# B&R Automation Studio project NewPendant_NG4_11_05_25A (part 19)

```c
					TVL_ROT_Param_Set[i].pEncoder = &AxisCh[TML_AX_TVL].curPos;
					TVL_ROT_Param_Set[i].pHomePos = &OLD_MTR_POS[TVL_ENC_HOME];
					TVL_ROT_Param_Set[i].EncPerTick = m->pCfg->HeadCfg.TVL.EncPerTick;
					TVL_ROT_Param_Set[i].EncDir = m->pCfg->HeadCfg.TVL.Enc_Dir;
					TVL_ROT_Param_Set[i].TicksAtHighVel = 3;

				break;

			}
		}

		for(i=0 ; i < 1 ; i++){

			switch(i){

				case 0:

					strcpy(Process[m->pCfg->HeadCfg.INDX.PROC_Indx].Name , "INDX");
					INDEX_Param_Set[i].pPrc = &Process[m->pCfg->HeadCfg.INDX.PROC_Indx];
					Process[m->pCfg->HeadCfg.INDX.PROC_Indx].Disable = 1;

				break;

			}

		}

	return 1;

}

DINT Configure_OMEGA_16INCH_HP_ENCODER(MASTER_typ *m  , UINT headType ){

}

/////////////////////////////////////////////////////////////

void ParametrAssignToPointers(MASTER_typ *m  , UINT indx){
int i;
CurCfg_typ *c;
Cfg_typ *cfg;
CurCalib_typ *calib;
DINT headType;

	if(!m)
		return;

	if(!m->pCurCfg)
		return;

	if(!m->pCalib)
		return;

	if(!m->pCalib->GenSetup)
		return;

	if(!m->pCfg)
		return;

	cfg = m->pCfg;

	c = m->pCurCfg;

	 headType = m->pCalib->GenSetup[SETUP_HEAD_SETUP];

	for(i=0 ; i < 1; i++){

		switch(i){

			case 0:

				//strcpy(Process[PROC_TIG_PS].Name , "TIG PS");

				if(c->Param[parTIG_StartDly].segmYes)
						PS_Param_Set[i].pStartDly		= &c->Param[parTIG_StartDly].val[indx];
				else 	PS_Param_Set[i].pStartDly		= &c->Param[parTIG_StartDly].val[0];

				if(c->Param[parTIG_StopDly].segmYes)
						PS_Param_Set[i].pStopDly		= &c->Param[parTIG_StopDly].val[indx];
				else		PS_Param_Set[i].pStopDly		= &c->Param[parTIG_StopDly].val[0];

				if(c->Param[parTIG_RampUp].segmYes)
						PS_Param_Set[i].pRampUp			= &c->Param[parTIG_RampUp].val[indx];
				else		PS_Param_Set[i].pRampUp			= &c->Param[parTIG_RampUp].val[0];

				if(c->Param[parTIG_RampDwn].segmYes)
						PS_Param_Set[i].pRampDwn		= &c->Param[parTIG_RampDwn].val[indx];
				else	PS_Param_Set[i].pRampDwn		= &c->Param[parTIG_RampDwn].val[0];

				if(c->Param[parTIG_AmpSP].segmYes)
						PS_Param_Set[i].pAmpSP			= &c->Param[parTIG_AmpSP].val[indx];
				else	PS_Param_Set[i].pAmpSP			= &c->Param[parTIG_AmpSP].val[0];

				if(c->Param[parTIG_AmpInSP].segmYes)
						PS_Param_Set[i].pAmpInSP		= &c->Param[parTIG_AmpInSP].val[indx];
				else	PS_Param_Set[i].pAmpInSP		= &c->Param[parTIG_AmpInSP].val[0];

				if(c->Param[parTIG_AmpOutSP].segmYes)
						PS_Param_Set[i].pAmpOutSP		= &c->Param[parTIG_AmpOutSP].val[indx];
				else	PS_Param_Set[i].pAmpOutSP		= &c->Param[parTIG_AmpOutSP].val[0];

				if(c->Param[parTIG_BackAmp].segmYes)
						PS_Param_Set[i].pBackAmp		= &c->Param[parTIG_BackAmp].val[indx];
				else		PS_Param_Set[i].pBackAmp 		= &c->Param[parTIG_BackAmp].val[0];

				if(c->Param[parTIG_StartAmp].segmYes)
						PS_Param_Set[i].pStartAmp		= &c->Param[parTIG_StartAmp].val[indx];
				else		PS_Param_Set[i].pStartAmp		= &c->Param[parTIG_StartAmp].val[0];

				if(c->Param[parTIG_EndAmp].segmYes)
						PS_Param_Set[i].pEndAmp			= &c->Param[parTIG_EndAmp].val[indx];
				else		PS_Param_Set[i].pEndAmp			= &c->Param[parTIG_EndAmp].val[0];

				if(c->Param[parTIG_AmpSP_Boost].segmYes)
						PS_Param_Set[i].pAmpBoost 		= &c->Param[parTIG_AmpSP_Boost].val[indx];
				else	PS_Param_Set[i].pAmpBoost 			= &c->Param[parTIG_AmpSP_Boost].val[0];

				if(c->Param_ENUM[parENUM_TIG_Mode].segmYes)
						PS_Param_Set[i].pMode			= &c->Param_ENUM[parENUM_TIG_Mode].val[indx];
				else 	PS_Param_Set[i].pMode			= &c->Param_ENUM[parENUM_TIG_Mode].val[0];

				if(c->Param[parTIG_PulseFreq].segmYes)
						PS_Param_Set[i].pPulseFreq 		= &c->Param[parTIG_PulseFreq].val[indx];
				else		PS_Param_Set[i].pPulseFreq 		= &c->Param[parTIG_PulseFreq].val[0];

				if(c->Param[parTIG_PulseWidth].segmYes)
						PS_Param_Set[i].pPulseWidth 		= &c->Param[parTIG_PulseWidth].val[indx];
				else		PS_Param_Set[i].pPulseWidth 		= &c->Param[parTIG_PulseWidth].val[0];

				if(c->Param[parTIG_Boost1].segmYes)
						PS_Param_Set[i].pBoost1 		= &c->Param[parTIG_Boost1].val[indx];
				else	PS_Param_Set[i].pBoost1 		= &c->Param[parTIG_Boost1].val[0];

				if(c->Param[parTIG_Boost2].segmYes)
						PS_Param_Set[i].pBoost2 		= &c->Param[parTIG_Boost2].val[indx];
				else	PS_Param_Set[i].pBoost2 		= &c->Param[parTIG_Boost2].val[0];

				if(c->Param[parCONTIN_TIG_RampDwn].segmYes)
						PS_Param_Set[i].pContin_RampDwn 		= &c->Param[parCONTIN_TIG_RampDwn].val[indx];
				else	PS_Param_Set[i].pContin_RampDwn 		= &c->Param[parCONTIN_TIG_RampDwn].val[0];

				if(c->Param[parCONTIN_TIG_RampUp].segmYes)
						PS_Param_Set[i].pContin_RampUp 		= &c->Param[parCONTIN_TIG_RampUp].val[indx];
				else	PS_Param_Set[i].pContin_RampUp 		= &c->Param[parCONTIN_TIG_RampUp].val[0];

				if(c->Param[parCONTIN_TIG_Dwell].segmYes)
						PS_Param_Set[i].pContin_Dwell 		= &c->Param[parCONTIN_TIG_Dwell].val[indx];
				else	PS_Param_Set[i].pContin_Dwell 		= &c->Param[parCONTIN_TIG_Dwell].val[0];

				if(c->Param[parCONTIN_TIG_Percent].segmYes)
						PS_Param_Set[i].pContin_Amp_Reduce 		= &c->Param[parCONTIN_TIG_Percent].val[indx];
				else	PS_Param_Set[i].pContin_Amp_Reduce 		= &c->Param[parCONTIN_TIG_Percent].val[0];

			break;

		}

	}

	for(i=0 ; i < 1 ; i++){

		switch(i){

			case 0:

				strcpy(Process[PROC_AVC].Name , "AVC");

				if(c->Param[parAVC_TouchVolt].segmYes)
						AVC_Param_Set[i].pTouchVolt 		= &c->Param[parAVC_TouchVolt].val[indx];
				else 	AVC_Param_Set[i].pTouchVolt 		= &c->Param[parAVC_TouchVolt].val[0];

				if(c->Param[parAVC_TouchTm].segmYes)
						AVC_Param_Set[i].pTouchTm 			= &c->Param[parAVC_TouchTm].val[indx];
				else 	AVC_Param_Set[i].pTouchTm 			= &c->Param[parAVC_TouchTm].val[0];

				if(c->Param[parAVC_TRetractTm].segmYes)
						AVC_Param_Set[i].pRetractTm 		= &c->Param[parAVC_TRetractTm].val[indx];
				else 	AVC_Param_Set[i].pRetractTm 		= &c->Param[parAVC_TRetractTm].val[0];

				if(c->Param[parAVC_TouchRepeat].segmYes)
						AVC_Param_Set[i].pTouchRepeat 		= &c->Param[parAVC_TouchRepeat].val[indx];
				else 	AVC_Param_Set[i].pTouchRepeat 		= &c->Param[parAVC_TouchRepeat].val[0];

				if(c->Param[parAVC_VoltSP].segmYes)
						AVC_Param_Set[i].pVoltSP 			= &c->Param[parAVC_VoltSP].val[indx];
				else 	AVC_Param_Set[i].pVoltSP 			= &c->Param[parAVC_VoltSP].val[0];

				if(c->Param[parAVC_VoltInSP].segmYes)
						AVC_Param_Set[i].pVoltInSP 			= &c->Param[parAVC_VoltInSP].val[indx];
				else 	AVC_Param_Set[i].pVoltInSP 			= &c->Param[parAVC_VoltInSP].val[0];

				if(c->Param[parAVC_VoltOutSP].segmYes)
						AVC_Param_Set[i].pVoltOutSP 		= &c->Param[parAVC_VoltOutSP].val[indx];
				else 	AVC_Param_Set[i].pVoltOutSP 		= &c->Param[parAVC_VoltOutSP].val[0];

				if(c->Param[parAVC_VoltBackSP].segmYes)
						AVC_Param_Set[i].pBkgVoltSP			= &c->Param[parAVC_VoltBackSP].val[indx];
				else 	AVC_Param_Set[i].pBkgVoltSP 		= &c->Param[parAVC_VoltBackSP].val[0];

				if(c->Param[parAVC_VSPTmOut].segmYes)
						AVC_Param_Set[i].pVoltSPTimeOut 	= &c->Param[parAVC_VSPTmOut].val[indx];
				else 	AVC_Param_Set[i].pVoltSPTimeOut 	= &c->Param[parAVC_VSPTmOut].val[0];

				if(c->Param[parAVC_TouchVel].segmYes)
						AVC_Param_Set[i].pTouchVel 			= &c->Param[parAVC_TouchVel].val[indx];
				else 	AVC_Param_Set[i].pTouchVel 			= &c->Param[parAVC_TouchVel].val[0];

				if(c->Param[parAVC_ToSPVel].segmYes)
						AVC_Param_Set[i].pToSPVel 			= &c->Param[parAVC_ToSPVel].val[indx];
				else 	AVC_Param_Set[i].pToSPVel 			= &c->Param[parAVC_ToSPVel].val[0];

				if(c->Param[parAVC_LU_TM].segmYes)
						AVC_Param_Set[i].pLU_Tm 			= &c->Param[parAVC_LU_TM].val[indx];
				else 	AVC_Param_Set[i].pLU_Tm 			= &c->Param[parAVC_LU_TM].val[0];

				if(c->Param[parAVC_KissTm].segmYes)
						AVC_Param_Set[i].pKiss_Tm 			= &c->Param[parAVC_KissTm].val[indx];
				else 	AVC_Param_Set[i].pKiss_Tm 			= &c->Param[parAVC_KissTm].val[0];

				if(c->Param[parAVC_VoltFinal].segmYes)
						AVC_Param_Set[i].pFinalVolt 		= &c->Param[parAVC_VoltFinal].val[indx];
				else 	AVC_Param_Set[i].pFinalVolt 		= &c->Param[parAVC_VoltFinal].val[0];

				if(c->Param[parAVC_DownSlope].segmYes)
						AVC_Param_Set[i].pRampDwn 		= &c->Param[parAVC_DownSlope].val[indx];
				else 	AVC_Param_Set[i].pRampDwn 		= &c->Param[parAVC_DownSlope].val[0];

				if(c->Param[parAVC_HoldTm].segmYes)
						AVC_Param_Set[i].pHoldTm 			= &c->Param[parAVC_HoldTm].val[indx];
				else 	AVC_Param_Set[i].pHoldTm 			= &c->Param[parAVC_HoldTm].val[0];

				if(c->Param[parAVC_GoBackTm].segmYes)
						AVC_Param_Set[i].pGoBackTm 			= &c->Param[parAVC_GoBackTm].val[indx];
				else 	AVC_Param_Set[i].pGoBackTm 			= &c->Param[parAVC_GoBackTm].val[0];

				if(c->Param[parAVC_StartDly].segmYes)
						AVC_Param_Set[i].pStartDly 			= &c->Param[parAVC_StartDly].val[indx];
				else 	AVC_Param_Set[i].pStartDly 			= &c->Param[parAVC_StartDly].val[0];

				if(c->Param[parAVC_StopDly].segmYes)
						AVC_Param_Set[i].pStopDly			= &c->Param[parAVC_StopDly].val[indx];
				else 	AVC_Param_Set[i].pStopDly 			= &c->Param[parAVC_StopDly].val[0];

				if(c->Param[parAVC_VoltInit].segmYes)
						AVC_Param_Set[i].pVoltInit			= &c->Param[parAVC_VoltInit].val[indx];
				else 	AVC_Param_Set[i].pVoltInit 			= &c->Param[parAVC_VoltInit].val[0];

				if(c->Param[parAVC_Upslope].segmYes)
						AVC_Param_Set[i].pRampUp 			= &c->Param[parAVC_Upslope].val[indx];
				else 	AVC_Param_Set[i].pRampUp 			= &c->Param[parAVC_Upslope].val[0];

				if(c->Param[parAVC_MaxVoltError].segmYes)
						AVC_Param_Set[i].pMaxVolrError 		= &c->Param[parAVC_MaxVoltError].val[indx];
				else 	AVC_Param_Set[i].pMaxVolrError 		= &c->Param[parAVC_MaxVoltError].val[0];

				if(c->Param[parAVC_Limits_Mask_Tm].segmYes)
						AVC_Param_Set[i].pLimitsFilterTm 	= &c->Param[parAVC_Limits_Mask_Tm].val[indx];
				else 	AVC_Param_Set[i].pLimitsFilterTm 	= &c->Param[parAVC_Limits_Mask_Tm].val[0];

				if(c->Param[parAVC_JogSpeedDirCntrl].segmYes)
						AVC_Param_Set[i].pJogSpeedDirCntrl	= &c->Param[parAVC_JogSpeedDirCntrl].val[indx];
				else 	AVC_Param_Set[i].pJogSpeedDirCntrl	= &c->Param[parAVC_JogSpeedDirCntrl].val[0];

				if(c->Param[parAVC_LiftSpeedDirCntrl].segmYes)
						AVC_Param_Set[i].pLiftSpeedDirCntrl	= &c->Param[parAVC_LiftSpeedDirCntrl].val[indx];
				else 	AVC_Param_Set[i].pLiftSpeedDirCntrl	= &c->Param[parAVC_LiftSpeedDirCntrl].val[0];

				if(c->Param_ENUM[parENUM_AVC_Mode].segmYes)
						AVC_Param_Set[i].pMode				= &c->Param_ENUM[parENUM_AVC_Mode].val[indx];
				else 	AVC_Param_Set[i].pMode				= &c->Param_ENUM[parENUM_AVC_Mode].val[0];

				if(c->Param[parAVC_LiftSpeedDirCntrl].segmYes)
						AVC_Param_Set[i].pJogSpeedDirCntrl	= &c->Param[parAVC_JogSpeedDirCntrl].val[indx];
				else 	AVC_Param_Set[i].pJogSpeedDirCntrl	= &c->Param[parAVC_JogSpeedDirCntrl].val[0];

				if(c->Param[parAVC_DB_Window].segmYes)
						AVC_Param_Set[i].pBB_Window 	= &c->Param[parAVC_DB_Window].val[indx];
				else 	AVC_Param_Set[i].pBB_Window		= &c->Param[parAVC_DB_Window].val[0];

				if(c->Param[parAVC_BB_Vel].segmYes)
						AVC_Param_Set[i].pBB_Vel		= &c->Param[parAVC_BB_Vel].val[indx];
				else 	AVC_Param_Set[i].pBB_Vel 	= &c->Param[parAVC_BB_Vel].val[0];

				if(c->Param[parAVC_BB_Gain].segmYes)
						AVC_Param_Set[i].pBB_Gain	= &c->Param[parAVC_BB_Gain].val[indx];
				else 	AVC_Param_Set[i].pBB_Gain 	= &c->Param[parAVC_BB_Gain].val[0];

				if(c->Param[parAVC_BB_Integr].segmYes)
						AVC_Param_Set[i].pBB_Integr	= &c->Param[parAVC_BB_Integr].val[indx];
				else 	AVC_Param_Set[i].pBB_Integr 	= &c->Param[parAVC_BB_Integr].val[0];

				if(c->Param[parAVC_Boost1].segmYes)
						AVC_Param_Set[i].pBoost1	= &c->Param[parAVC_Boost1].val[indx];
				else 	AVC_Param_Set[i].pBoost1 	= &c->Param[parAVC_Boost1].val[0];

				if(c->Param[parAVC_Boost2].segmYes)
						AVC_Param_Set[i].pBoost2	= &c->Param[parAVC_Boost2].val[indx];
				else 	AVC_Param_Set[i].pBoost2 	= &c->Param[parAVC_Boost2].val[0];

			break;

		}
	}

	for(i=0 ; i < 1 ; i++){

		switch(i){

			case 0:

				if(c->Param[parWRST_JogSpeedDirCntrl].segmYes)
						WRST_TML_Param_Set[i].pJogSpeedDirCntrl		= &c->Param[parWRST_JogSpeedDirCntrl].val[indx];
				else 	WRST_TML_Param_Set[i].pJogSpeedDirCntrl		= &c->Param[parWRST_JogSpeedDirCntrl].val[0];

				if(c->Param[parTVL_POS_OFFSET].segmYes)
						WRST_TML_Param_Set[i].pTVL_Pos_Offset 	= &c->Param[parTVL_POS_OFFSET].val[indx];
				else	WRST_TML_Param_Set[i].pTVL_Pos_Offset 	= &c->Param[parTVL_POS_OFFSET].val[0];

				if(c->Param[parTVL_POS_PREDICT].segmYes)
						WRST_TML_Param_Set[i].pTVL_Pos_Predict 	= &c->Param[parTVL_POS_PREDICT].val[indx];
				else	WRST_TML_Param_Set[i].pTVL_Pos_Predict 	= &c->Param[parTVL_POS_PREDICT].val[0];

				if(c->Param[parGEN_Radius].segmYes)
						WRST_TML_Param_Set[i].pRadius		= &c->Param[parGEN_Radius].val[indx];
				else 	WRST_TML_Param_Set[i].pRadius		= &c->Param[parGEN_Radius].val[0];

				if(c->Param[parGEN_RadSpeed_Boost].segmYes)
						WRST_TML_Param_Set[i].pRadSpeed_Boost		= &c->Param[parGEN_RadSpeed_Boost].val[indx];
				else 	WRST_TML_Param_Set[i].pRadSpeed_Boost		= &c->Param[parGEN_RadSpeed_Boost].val[0];

			break;

		}
	}

	for(i=0 ; i < 1 ; i++){

		switch(i){

			case 0:

				strcpy(Process[PROC_OSC].Name , "OSC");

				if(c->Param[parOSC_StartDly].segmYes)
						OSC_TML_Param_Set[i].pStartDly		= &c->Param[parOSC_StartDly].val[indx];
				else 	OSC_TML_Param_Set[i].pStartDly		= &c->Param[parOSC_StartDly].val[0];

				if(c->Param[parOSC_RampUp].segmYes)
						OSC_TML_Param_Set[i].pRampUp		= &c->Param[parOSC_RampUp].val[indx];
				else 	OSC_TML_Param_Set[i].pRampUp		= &c->Param[parOSC_RampUp].val[0];

				if(c->Param[parOSC_Amplit].segmYes)
						OSC_TML_Param_Set[i].pPrimAmpl		= &c->Param[parOSC_Amplit].val[indx];
				else 	OSC_TML_Param_Set[i].pPrimAmpl		= &c->Param[parOSC_Amplit].val[0];

				if(c->Param[parOSC_InitAmplit].segmYes)
						OSC_TML_Param_Set[i].pInitAmpl		= &c->Param[parOSC_InitAmplit].val[indx];
				else	OSC_TML_Param_Set[i].pInitAmpl		= &c->Param[parOSC_InitAmplit].val[0];

				if(c->Param[parOSC_FinalAmplit].segmYes)
						OSC_TML_Param_Set[i].pFinalAmpl		= &c->Param[parOSC_FinalAmplit].val[indx];
				else	OSC_TML_Param_Set[i].pFinalAmpl		= &c->Param[parOSC_FinalAmplit].val[0];

				if(c->Param[parOSC_StopDly].segmYes)
						OSC_TML_Param_Set[i].pStopDly		= &c->Param[parOSC_StopDly].val[indx];
				else 	OSC_TML_Param_Set[i].pStopDly		= &c->Param[parOSC_StopDly].val[0];

				if(c->Param[parOSC_RampDwn].segmYes)
						OSC_TML_Param_Set[i].pRampDwn		= &c->Param[parOSC_RampDwn].val[indx];
				else 	OSC_TML_Param_Set[i].pRampDwn		= &c->Param[parOSC_RampDwn].val[0];

				if(c->Param[parOSC_RampUpdate].segmYes)
						OSC_TML_Param_Set[i].pRampUpdate	= &c->Param[parOSC_RampUpdate].val[indx];
				else 	OSC_TML_Param_Set[i].pRampUpdate	= &c->Param[parOSC_RampUpdate].val[0];

				if(c->Param[parOSC_Excur].segmYes)
						OSC_TML_Param_Set[i].pFreq			= &c->Param[parOSC_Excur].val[indx];
				else 	OSC_TML_Param_Set[i].pFreq			= &c->Param[parOSC_Excur].val[0];

				if(cfg->HeadCfg.OSC.DwellDir > 0){

					if(c->Param[parOSC_Dwell_In].segmYes)
						OSC_TML_Param_Set[i].pDwell_In		= &c->Param[parOSC_Dwell_Out].val[indx];
					else	OSC_TML_Param_Set[i].pDwell_In		= &c->Param[parOSC_Dwell_Out].val[0];

					if(c->Param[parOSC_Dwell_Out].segmYes)
						OSC_TML_Param_Set[i].pDwell_Out 	= &c->Param[parOSC_Dwell_In].val[indx];
					else	OSC_TML_Param_Set[i].pDwell_Out 	= &c->Param[parOSC_Dwell_In].val[0];

				}
				else {

					if(c->Param[parOSC_Dwell_In].segmYes)
							OSC_TML_Param_Set[i].pDwell_In		= &c->Param[parOSC_Dwell_In].val[indx];
					else	OSC_TML_Param_Set[i].pDwell_In		= &c->Param[parOSC_Dwell_In].val[0];

					if(c->Param[parOSC_Dwell_Out].segmYes)
							OSC_TML_Param_Set[i].pDwell_Out 	= &c->Param[parOSC_Dwell_Out].val[indx];
					else	OSC_TML_Param_Set[i].pDwell_Out 	= &c->Param[parOSC_Dwell_Out].val[0];

				}

				if(c->Param_ENUM[parENUM_OSC_CAM].segmYes)
						OSC_TML_Param_Set[i].pCamType		= &c->Param_ENUM[parENUM_OSC_CAM].val[indx];
				else 	OSC_TML_Param_Set[i].pCamType		= &c->Param_ENUM[parENUM_OSC_CAM].val[0];

				if(c->Param[parOSC_JogSpeed].segmYes)
						OSC_TML_Param_Set[i].pJogSpeed		= &c->Param[parOSC_JogSpeed].val[indx];
				else 	OSC_TML_Param_Set[i].pJogSpeed		= &c->Param[parOSC_JogSpeed].val[0];

				if(c->Param[parOSC_JogSpeedDirCntrl].segmYes)
						OSC_TML_Param_Set[i].pJogSpeedDirCntrl		= &c->Param[parOSC_JogSpeedDirCntrl].val[indx];
				else 	OSC_TML_Param_Set[i].pJogSpeedDirCntrl		= &c->Param[parOSC_JogSpeedDirCntrl].val[0];

				////

				if(c->Param_ENUM[parENUM_OSC_Mode].segmYes)
						OSC_TML_Param_Set[i].pOSC_Mode		= &c->Param_ENUM[parENUM_OSC_Mode].val[indx];
				else 	OSC_TML_Param_Set[i].pOSC_Mode		= &c->Param_ENUM[parENUM_OSC_Mode].val[0];

				if(c->Param_ENUM[parENUM_OSC_Synch].segmYes)
						OSC_TML_Param_Set[i].pOSC_Synch		= &c->Param_ENUM[parENUM_OSC_Synch].val[indx];
				else	OSC_TML_Param_Set[i].pOSC_Synch		= &c->Param_ENUM[parENUM_OSC_Synch].val[0];

				if(c->Param[parOSC_Indx].segmYes)
						OSC_TML_Param_Set[i].pIndexDist		= &c->Param[parOSC_Indx].val[indx];
				else	OSC_TML_Param_Set[i].pIndexDist		= &c->Param[parOSC_Indx].val[0];

				if(c->Param[parOSC_Period].segmYes)
						OSC_TML_Param_Set[i].pPeriod		= &c->Param[parOSC_Period].val[indx];
				else	OSC_TML_Param_Set[i].pPeriod		= &c->Param[parOSC_Period].val[0];

				if(c->Param[parOSC_Indx_Vel].segmYes)
						OSC_TML_Param_Set[i].pIndxVel		= &c->Param[parOSC_Indx_Vel].val[indx];
				else	OSC_TML_Param_Set[i].pIndxVel		= &c->Param[parOSC_Indx_Vel].val[0];

			break;

		}

	}

	for(i=0 ; i < 1 ; i++){

		switch(i){

			case 0:

				strcpy(Process[PROC_GAS].Name , "GAS");

				if(c->Param[parGAS_PrePurgeTm].segmYes)
						GAS_Param_Set[i].pStartDly		= &c->Param[parGAS_PrePurgeTm].val[indx];
				else 	GAS_Param_Set[i].pStartDly		= &c->Param[parGAS_PrePurgeTm].val[0];

				if(c->Param[parGAS_PostPurgeTm].segmYes)
						GAS_Param_Set[i].pStopDly		= &c->Param[parGAS_PostPurgeTm].val[indx];
				else 	GAS_Param_Set[i].pStopDly		= &c->Param[parGAS_PostPurgeTm].val[0];

				if(c->Param[parGAS_Tmo].segmYes)
						GAS_Param_Set[i].pTmo			= &c->Param[parGAS_Tmo].val[indx];
				else 	GAS_Param_Set[i].pTmo			= &c->Param[parGAS_Tmo].val[0];

			break;

		}

	}

	for(i=0 ; i < 1 ; i++){

		switch(i){

			case 0:

				strcpy(Process[PROC_INDX].Name , "INDX");

				if(c->Param[parINDX_StepDist].segmYes)
						INDEX_Param_Set[i].pStepDist		= &c->Param[parINDX_StepDist].val[indx];
				else	INDEX_Param_Set[i].pStepDist		= &c->Param[parINDX_StepDist].val[0];

				if(c->Param[parINDX_StepVel].segmYes)
						INDEX_Param_Set[i].pStepVel		= &c->Param[parINDX_StepVel].val[indx];
				else	INDEX_Param_Set[i].pStepVel		= &c->Param[parINDX_StepVel].val[0];

				if(c->Param[parINDX_JogSpeedDirCntrl].segmYes)
						INDEX_Param_Set[i].pJogSpeedDirCntrl = &c->Param[parINDX_JogSpeedDirCntrl].val[indx];
				else	INDEX_Param_Set[i].pJogSpeedDirCntrl = &c->Param[parINDX_JogSpeedDirCntrl].val[0];

			break;

		}

	}

	for(i=0 ; i < 1; i++){

		switch(i){

			case 0:

				strcpy(Process[PROC_COOL].Name , "COOLANT");

				if(c->Param[parCOOL_Tmo].segmYes)
						COOL_Param_Set[i].pTmo = &c->Param[parCOOL_Tmo].val[indx];
				else 	COOL_Param_Set[i].pTmo = &c->Param[parCOOL_Tmo].val[0];

			break;

		}

	}

	for(i=0 ; i < 1; i++){

		switch(i){

			case 0:

				strcpy(Process[PROC_HW_PS].Name , "HW PS");

				if(c->Param[parHW_RampDwnDly].segmYes)
						HW_PS_Param_Set[i].pStartDly	= &c->Param[parHW_RampDwnDly].val[indx];
				else 	HW_PS_Param_Set[i].pStartDly	= &c->Param[parHW_RampDwnDly].val[0];

				if(c->Param[parHW_RampDwnDly].segmYes)
						HW_PS_Param_Set[i].pStopDly 	= &c->Param[parHW_RampDwnDly].val[indx];
				else 	HW_PS_Param_Set[i].pStopDly 	= &c->Param[parHW_RampDwnDly].val[0];

				if(c->Param[parHW_RampUp].segmYes)
						HW_PS_Param_Set[i].pRampUp		= &c->Param[parHW_RampUp].val[indx];
				else 	HW_PS_Param_Set[i].pRampUp		= &c->Param[parHW_RampUp].val[0];

				if(c->Param[parHW_RampDwn].segmYes)
						HW_PS_Param_Set[i].pRampDwn 	= &c->Param[parHW_RampDwn].val[indx];
				else 	HW_PS_Param_Set[i].pRampDwn 	= &c->Param[parHW_RampDwn].val[0];

				if(c->Param[parHW_StartAmp].segmYes)
						HW_PS_Param_Set[i].pStartAmp	= &c->Param[parHW_StartAmp].val[indx];
				else 	HW_PS_Param_Set[i].pStartAmp	= &c->Param[parHW_StartAmp].val[0];

				if(c->Param[parHW_AmpSP].segmYes)
						HW_PS_Param_Set[i].pAmpSP		= &c->Param[parHW_AmpSP].val[indx];
				else 	HW_PS_Param_Set[i].pAmpSP		= &c->Param[parHW_AmpSP].val[0];

				if(c->Param[parHW_EndAmp].segmYes)
						HW_PS_Param_Set[i].pEndAmp		= &c->Param[parHW_EndAmp].val[indx];
				else 	HW_PS_Param_Set[i].pEndAmp		= &c->Param[parHW_EndAmp].val[0];

				if(c->Param[parHW_RampUpdate].segmYes)
						HW_PS_Param_Set[i].pRampUpdate 	= &c->Param[parHW_RampUpdate].val[indx];
				else 	HW_PS_Param_Set[i].pRampUpdate 	= &c->Param[parHW_RampUpdate].val[0];

				if(c->Param[parHW_VoltSP].segmYes)
						HW_PS_Param_Set[i].pVoltSP 		= &c->Param[parHW_VoltSP].val[indx];
				else 	HW_PS_Param_Set[i].pVoltSP		= &c->Param[parHW_VoltSP].val[0];

				if(c->Param[parHW_AmpSP_Boost].segmYes)
						HW_PS_Param_Set[i].pAmpBoost 	= &c->Param[parHW_AmpSP_Boost].val[indx];
				else 	HW_PS_Param_Set[i].pAmpBoost 	= &c->Param[parHW_AmpSP_Boost].val[0];

			break;

		}

	}

	for(i=0 ; i < 2; i++){

		switch(i){

			case 0:

				if(i == 0)
					strcpy(Process[PROC_WIRE_FEED].Name ,"WrFeed");
				else
					strcpy(Process[PROC_WIRE_FEED].Name ,"WrPulse");

				if(c->Param[parWF_StartDly].segmYes)
						WIRE_Param_Set[i].pStartDly		= &c->Param[parWF_StartDly].val[indx]; 			// 1
				else	WIRE_Param_Set[i].pStartDly		= &c->Param[parWF_StartDly].val[0];

				if(c->Param[parWF_SpeedSP].segmYes)
						WIRE_Param_Set[i].pSpeedSp		= &c->Param[parWF_SpeedSP].val[indx]; 			// 2
				else	WIRE_Param_Set[i].pSpeedSp		= &c->Param[parWF_SpeedSP].val[0];

				if(c->Param[parWF_SpeedInSP].segmYes)
						WIRE_Param_Set[i].pSpeedInSp		= &c->Param[parWF_SpeedInSP].val[indx]; 	// 3
				else	WIRE_Param_Set[i].pSpeedInSp		= &c->Param[parWF_SpeedInSP].val[0];

				if(c->Param[parWF_SpeedOutSP].segmYes)
						WIRE_Param_Set[i].pSpeedOutSp		= &c->Param[parWF_SpeedOutSP].val[indx]; 	// 4
				else	WIRE_Param_Set[i].pSpeedOutSp		= &c->Param[parWF_SpeedOutSP].val[0];

				if(c->Param[parWF_BkgSpeedSP].segmYes)
						WIRE_Param_Set[i].pBkgSpeedSp		= &c->Param[parWF_BkgSpeedSP].val[indx];	// 5
				else	WIRE_Param_Set[i].pBkgSpeedSp		= &c->Param[parWF_BkgSpeedSP].val[0];

				if(c->Param[parWF_SpeedInit].segmYes)
						WIRE_Param_Set[i].pSpeedInit	= &c->Param[parWF_SpeedInit].val[indx]; 		// 6
				else	WIRE_Param_Set[i].pSpeedInit	= &c->Param[parWF_SpeedInit].val[0];

				if(c->Param[parWF_SpeedFinal].segmYes)
						WIRE_Param_Set[i].pSpeedFinal	= &c->Param[parWF_SpeedFinal].val[indx]; 		// 7
				else	WIRE_Param_Set[i].pSpeedFinal	= &c->Param[parWF_SpeedFinal].val[0];

				if(c->Param[parWF_RampUp].segmYes)
						WIRE_Param_Set[i].pRampUp		= &c->Param[parWF_RampUp].val[indx]; 			// 8
				else	WIRE_Param_Set[i].pRampUp		= &c->Param[parWF_RampUp].val[0];

				if(c->Param[parWF_StopDly].segmYes)
						WIRE_Param_Set[i].pStopDly		= &c->Param[parWF_StopDly].val[indx]; 			// 9
				else	WIRE_Param_Set[i].pStopDly		= &c->Param[parWF_StopDly].val[0];

				if(c->Param[parWF_RampDwn].segmYes)
						WIRE_Param_Set[i].pRampDwn		= &c->Param[parWF_RampDwn].val[indx];			// 10
				else	WIRE_Param_Set[i].pRampDwn		= &c->Param[parWF_RampDwn].val[0];

				if(c->Param[parWF_RampUpdate].segmYes)
						WIRE_Param_Set[i].pRampUpdate	= &c->Param[parWF_RampUpdate].val[indx];		// 11
				else	WIRE_Param_Set[i].pRampUpdate	= &c->Param[parWF_RampUpdate].val[0];

				if(c->Param[parWF_Boost1SP].segmYes)
						WIRE_Param_Set[i].pBoost1SP		= &c->Param[parWF_Boost1SP].val[indx];			// 12
				else	WIRE_Param_Set[i].pBoost1SP		= &c->Param[parWF_Boost1SP].val[0];

				if(c->Param[parWF_Boost2SP].segmYes)
						WIRE_Param_Set[i].pBoost2SP		= &c->Param[parWF_Boost2SP].val[indx];			// 13
				else	WIRE_Param_Set[i].pBoost2SP		= &c->Param[parWF_Boost2SP].val[0];

				if(c->Param[parWF_JogSpeed].segmYes)
						WIRE_Param_Set[i].pJogSpeed		= &c->Param[parWF_JogSpeed].val[indx];			// 14
				else	WIRE_Param_Set[i].pJogSpeed		= &c->Param[parWF_JogSpeed].val[0];

				if(c->Param[parWF_JogSpeedDirCntrl].segmYes)
						WIRE_Param_Set[i].pJogSpeedDirCntrl	= &c->Param[parWF_JogSpeedDirCntrl].val[indx];	// 15
				else	WIRE_Param_Set[i].pJogSpeedDirCntrl	= &c->Param[parWF_JogSpeedDirCntrl].val[0];

				if(c->Param[parCONTIN_WF_RampDwn].segmYes)
						WIRE_Param_Set[i].pContinRampDwn		= &c->Param[parCONTIN_WF_RampDwn].val[indx];	// 16
				else	WIRE_Param_Set[i].pContinRampDwn    	= &c->Param[parCONTIN_WF_RampDwn].val[0];

				if(c->Param[parCONTIN_WF_RampUp].segmYes)
						WIRE_Param_Set[i].pContinRampUp		= &c->Param[parCONTIN_WF_RampUp].val[indx];		// 17
				else	WIRE_Param_Set[i].pContinRampUp    	= &c->Param[parCONTIN_WF_RampUp].val[0];

				//  Wire specific

				if(c->Param[parWF_RetractDly].segmYes)
						WIRE_Param_Set[i].pRetracDly		= &c->Param[parWF_RetractDly].val[indx];
				else	WIRE_Param_Set[i].pRetracDly		= &c->Param[parWF_RetractDly].val[0];

				if(c->Param[parWF_RetracDist].segmYes)
						WIRE_Param_Set[i].pRetracDist		= &c->Param[parWF_RetracDist].val[indx];
				else	WIRE_Param_Set[i].pRetracDist		= &c->Param[parWF_RetracDist].val[0];

				if(c->Param[parWF_RetractSpeed].segmYes)
						WIRE_Param_Set[i].pRetracSpeed		= &c->Param[parWF_RetractSpeed].val[indx];
				else	WIRE_Param_Set[i].pRetracSpeed		= &c->Param[parWF_RetractSpeed].val[0];

				if(c->Param_ENUM[parENUM_WF_AUX].segmYes)
						WIRE_Param_Set[i].pAuxMtrMode		= &c->Param_ENUM[parENUM_WF_AUX].val[indx];
				else 	WIRE_Param_Set[i].pAuxMtrMode		= &c->Param_ENUM[parENUM_WF_AUX].val[0];

				/*
				WIRE_Param_Set[i].pRetracDly = 0;
				WIRE_Param_Set[i].pRetracDist = 0;
				WIRE_Param_Set[i].pRetracSpeed = 0;
				WIRE_Param_Set[i].pAuxMtrMode = 0;
				*/

			break;

			case 1:

				strcpy(Process[PROC_WIRE_PULSE].Name ,"WrPulse");

				if(c->Param[parWP_StartDly].segmYes)
						WIRE_Param_Set[i].pStartDly		= &c->Param[parWP_StartDly].val[indx];    		// 1
				else	WIRE_Param_Set[i].pStartDly		= &c->Param[parWP_StartDly].val[0];

				if(c->Param[parWP_SpeedSP].segmYes)
						WIRE_Param_Set[i].pSpeedSp		= &c->Param[parWP_SpeedSP].val[indx];    		// 2
				else	WIRE_Param_Set[i].pSpeedSp		= &c->Param[parWP_SpeedSP].val[0];

				if(c->Param[parWP_SpeedInSP].segmYes)
						WIRE_Param_Set[i].pSpeedInSp		= &c->Param[parWP_SpeedInSP].val[indx]; 	// 3
				else	WIRE_Param_Set[i].pSpeedInSp		= &c->Param[parWP_SpeedInSP].val[0];

				if(c->Param[parWP_SpeedOutSP].segmYes)
						WIRE_Param_Set[i].pSpeedOutSp		= &c->Param[parWP_SpeedOutSP].val[indx];   	// 4
				else	WIRE_Param_Set[i].pSpeedOutSp		= &c->Param[parWP_SpeedOutSP].val[0];

				if(c->Param[parWP_BkgSpeedSP].segmYes)
						WIRE_Param_Set[i].pBkgSpeedSp		= &c->Param[parWP_BkgSpeedSP].val[indx]; 	// 5
				else	WIRE_Param_Set[i].pBkgSpeedSp		= &c->Param[parWP_BkgSpeedSP].val[0];

				if(c->Param[parWP_SpeedInit].segmYes)
						WIRE_Param_Set[i].pSpeedInit	= &c->Param[parWP_SpeedInit].val[indx]; 		// 6
				else	WIRE_Param_Set[i].pSpeedInit	= &c->Param[parWP_SpeedInit].val[0];

				if(c->Param[parWP_SpeedFinal].segmYes)
						WIRE_Param_Set[i].pSpeedFinal	= &c->Param[parWP_SpeedFinal].val[indx]; 		// 7
				else	WIRE_Param_Set[i].pSpeedFinal	= &c->Param[parWP_SpeedFinal].val[0];

				if(c->Param[parWP_RampUp].segmYes)
						WIRE_Param_Set[i].pRampUp		= &c->Param[parWP_RampUp].val[indx]; 			// 8
				else	WIRE_Param_Set[i].pRampUp		= &c->Param[parWP_RampUp].val[0];

				if(c->Param[parWP_StopDly].segmYes)
						WIRE_Param_Set[i].pStopDly		= &c->Param[parWP_StopDly].val[indx]; 			// 9
				else	WIRE_Param_Set[i].pStopDly		= &c->Param[parWP_StopDly].val[0];

				if(c->Param[parWP_RampDwn].segmYes)
						WIRE_Param_Set[i].pRampDwn		= &c->Param[parWP_RampDwn].val[indx];			// 10
				else	WIRE_Param_Set[i].pRampDwn		= &c->Param[parWP_RampDwn].val[0];

				if(c->Param[parWP_RampUpdate].segmYes)
						WIRE_Param_Set[i].pRampUpdate	= &c->Param[parWP_RampUpdate].val[indx];		// 11
				else	WIRE_Param_Set[i].pRampUpdate	= &c->Param[parWP_RampUpdate].val[0];

				if(c->Param[parWP_Boost1SP].segmYes)
						WIRE_Param_Set[i].pBoost1SP		= &c->Param[parWP_Boost1SP].val[indx];			// 12
				else	WIRE_Param_Set[i].pBoost1SP		= &c->Param[parWP_Boost1SP].val[0];

				if(c->Param[parWP_Boost2SP].segmYes)
						WIRE_Param_Set[i].pBoost2SP		= &c->Param[parWP_Boost2SP].val[indx];			// 13
				else	WIRE_Param_Set[i].pBoost2SP		= &c->Param[parWP_Boost2SP].val[0];

				if(c->Param[parWP_JogSpeed].segmYes)
						WIRE_Param_Set[i].pJogSpeed		= &c->Param[parWP_JogSpeed].val[indx];			// 14
				else	WIRE_Param_Set[i].pJogSpeed		= &c->Param[parWP_JogSpeed].val[0];

				if(c->Param[parWP_JogSpeedDirCntrl].segmYes)
						WIRE_Param_Set[i].pJogSpeedDirCntrl	= &c->Param[parWP_JogSpeedDirCntrl].val[indx];		// 15
				else	WIRE_Param_Set[i].pJogSpeedDirCntrl	= &c->Param[parWP_JogSpeedDirCntrl].val[0];

				if(c->Param[parCONTIN_WP_RampDwn].segmYes)
						WIRE_Param_Set[i].pContinRampDwn		= &c->Param[parCONTIN_WP_RampDwn].val[indx];	// 16
				else	WIRE_Param_Set[i].pContinRampDwn		= &c->Param[parCONTIN_WP_RampDwn].val[0];

				if(c->Param[parCONTIN_WP_RampUp].segmYes)
						WIRE_Param_Set[i].pContinRampUp 	= &c->Param[parCONTIN_WP_RampUp].val[indx];			// 17
				else	WIRE_Param_Set[i].pContinRampUp 	= &c->Param[parCONTIN_WP_RampUp].val[0];

			break;

		}

	}

	for(i=0 ; i < 1; i++){

		switch(i){

			case 0:

				strcpy(Process[PROC_TVL].Name , "TVL");

				if(c->Param[parTVL_InitVel].segmYes)
						TVL_ROT_Param_Set[i].pInitVel 		= &c->Param[parTVL_InitVel].val[indx];
				else 	TVL_ROT_Param_Set[i].pInitVel 		= &c->Param[parTVL_InitVel].val[0];

				if(c->Param[parTVL_VelSP].segmYes)
						TVL_ROT_Param_Set[i].pPrimVel		= &c->Param[parTVL_VelSP].val[indx];
				else	TVL_ROT_Param_Set[i].pPrimVel		= &c->Param[parTVL_VelSP].val[0];

				if(c->Param[parTVL_VelInSP].segmYes)
						TVL_ROT_Param_Set[i].pPrimInVel		= &c->Param[parTVL_VelInSP].val[indx];
				else	TVL_ROT_Param_Set[i].pPrimInVel		= &c->Param[parTVL_VelInSP].val[0];

				if(c->Param[parTVL_VelOutSP].segmYes)
						TVL_ROT_Param_Set[i].pPrimOutVel		= &c->Param[parTVL_VelOutSP].val[indx];
				else	TVL_ROT_Param_Set[i].pPrimOutVel		= &c->Param[parTVL_VelOutSP].val[0];

				if(c->Param[parTVL_VelBackSP].segmYes)
						TVL_ROT_Param_Set[i].pPrimBackVel		= &c->Param[parTVL_VelBackSP].val[indx];
				else	TVL_ROT_Param_Set[i].pPrimBackVel		= &c->Param[parTVL_VelBackSP].val[0];

				if(c->Param[parTVL_FinalVel].segmYes)
						TVL_ROT_Param_Set[i].pFinalVel		= &c->Param[parTVL_FinalVel].val[indx];
				else	TVL_ROT_Param_Set[i].pFinalVel		= &c->Param[parTVL_FinalVel].val[0];

				if(c->Param[parTVL_Jog2Stop].segmYes)
						TVL_ROT_Param_Set[i].pJog2Stop = &c->Param[parTVL_Jog2Stop].val[indx];
				else	TVL_ROT_Param_Set[i].pJog2Stop 		= &c->Param[parTVL_Jog2Stop].val[0];

				if(c->Param[parTVL_JogSpeedDirCntrl].segmYes)
						TVL_ROT_Param_Set[i].pJogSpeedDirCntrl	= &c->Param[parTVL_JogSpeedDirCntrl].val[indx];
				else	TVL_ROT_Param_Set[i].pJogSpeedDirCntrl	= &c->Param[parTVL_JogSpeedDirCntrl].val[0];

				if(c->Param[parTVL_StartDly].segmYes)
						TVL_ROT_Param_Set[i].pStartDly 		= &c->Param[parTVL_StartDly].val[indx];
				else 	TVL_ROT_Param_Set[i].pStartDly 		= &c->Param[parTVL_StartDly].val[0];

				if(c->Param[parTVL_RampUp].segmYes)
						TVL_ROT_Param_Set[i].pRampUp		= &c->Param[parTVL_RampUp].val[indx];
				else 	TVL_ROT_Param_Set[i].pRampUp		= &c->Param[parTVL_RampUp].val[0];

				if(c->Param[parTVL_StopDly].segmYes)
						TVL_ROT_Param_Set[i].pStopDly		= &c->Param[parTVL_StopDly].val[indx];
				else 	TVL_ROT_Param_Set[i].pStopDly		= &c->Param[parTVL_StopDly].val[0];

				if(c->Param[parTVL_RampDwn].segmYes)
						TVL_ROT_Param_Set[i].pRampDwn		= &c->Param[parTVL_RampDwn].val[indx];
				else 	TVL_ROT_Param_Set[i].pRampDwn		= &c->Param[parTVL_RampDwn].val[0];

				if(c->Param[parTVL_RampUpdate].segmYes)
						TVL_ROT_Param_Set[i].pRampUpdate	= &c->Param[parTVL_RampUpdate].val[indx];
				else 	TVL_ROT_Param_Set[i].pRampUpdate	= &c->Param[parTVL_RampUpdate].val[0];

				if(c->Param[parTVL_RewrapDly].segmYes)
						TVL_ROT_Param_Set[i].pRewrapDly		= &c->Param[parTVL_RewrapDly].val[indx];
				else 	TVL_ROT_Param_Set[i].pRewrapDly		= &c->Param[parTVL_RewrapDly].val[0];

				if(c->Param[parTVL_RewrapVel].segmYes)
						TVL_ROT_Param_Set[i].pRewrapVel		= &c->Param[parTVL_RewrapVel].val[indx];
				else 	TVL_ROT_Param_Set[i].pRewrapVel		= &c->Param[parTVL_RewrapVel].val[0];

				if(c->Param[parTVL_Boost1].segmYes)
						TVL_ROT_Param_Set[i].pBoost1		= &c->Param[parTVL_Boost1].val[indx];
				else 	TVL_ROT_Param_Set[i].pBoost1		= &c->Param[parTVL_Boost1].val[0];

				if(c->Param[parTVL_Boost2].segmYes)
						TVL_ROT_Param_Set[i].pBoost2		= &c->Param[parTVL_Boost2].val[indx];
				else	TVL_ROT_Param_Set[i].pBoost2		= &c->Param[parTVL_Boost2].val[0];

				if(c->Param[parCONTIN_TVL_RampDwn].segmYes)
						TVL_ROT_Param_Set[i].pContinRampDwn		= &c->Param[parCONTIN_TVL_RampDwn].val[indx];
				else	TVL_ROT_Param_Set[i].pContinRampDwn		= &c->Param[parCONTIN_TVL_RampDwn].val[0];

				if(c->Param[parCONTIN_TVL_RampUp].segmYes)
						TVL_ROT_Param_Set[i].pContinRampUp		= &c->Param[parCONTIN_TVL_RampUp].val[indx];
				else	TVL_ROT_Param_Set[i].pContinRampUp		= &c->Param[parCONTIN_TVL_RampUp].val[0];

			break;

		}

	}

}

DINT NextDivider(DINT *in , DINT mod , BOOL dir){
DINT x , base;

/*
return :

-1 ->  wrong module
0 -> not exists counting up
1 -> not exist counting down
2 -> OK found

*/

	x = *in;
	base = *in;

	if(mod < 1){
		*in = 1;
		return -1;

	}

	if(dir){

		do{

			x++;

			if(x > mod){

				*in = mod;
				return 0;

			}

		}while( remainderf ((float)mod,(float)x));

	}
	else{

		do{
			x--;

			if(x < 1){
				*in = 1;
				return 1;

			}

		}while( remainderf ((float)mod,(float)x));
	}

	*in = x;
	return 2;

}

DINT PickPinsNo(DINT *indx , DINT mod  ){
int i;
DINT x , ret;

	x = 1;

	if(mod < 1)
		return -100;

	if(*indx >= 0){

		for(i = 0 ; i < *indx ; i++){

			if( NextDivider(&x , mod , 1)== 0 ){

				ret = mod/x;
				*indx = i;
				return ret;// max indx

			}

		}

	}
	else{

		ret = mod;
		*indx = 0;
		return ret; // min indx

	}

	ret = mod/x;
	return ret;

}

void PleaseUpdateHeadSetup(MASTER_typ *m ){
DINT x , k;

CurCalib_typ *curCalib ;
CurCfg_typ *curCfg;

INT pinsPerZone;

	if(!m)
		return;

	curCalib = m->pCalib;
	curCfg	 = m->pCurCfg;

	if(!curCalib || !curCfg)
		return;

	if(curCalib->GenSetup[SETUP_PIN_PER_ROT]< 1)
		curCalib->GenSetup[SETUP_PIN_PER_ROT] = 1;

	////////////////////////////////////////////////////////////
	//  Calculate number of Segment and Zone
	curCalib->GenSetup[SETUP_SEGM_NO] = curCalib->GenSetup[SETUP_PIN_PER_ROT] ;
	m->ticksPerSegm = 1;
	m->numSegm = curCalib->GenSetup[SETUP_PIN_PER_ROT] / m->ticksPerSegm;

	if(curCfg->Param_INT[parINT_NumZone].val[0]> 32.0)
		curCfg->Param_INT[parINT_NumZone].val[0] = 32.0;

	if(curCfg->Param_INT[parINT_NumZone].val[0]> (float)curCalib->GenSetup[SETUP_PIN_PER_ROT])
		curCfg->Param_INT[parINT_NumZone].val[0] = (float)curCalib->GenSetup[SETUP_PIN_PER_ROT];

	if(curCfg->Param_INT[parINT_NumZone].val[0]< 1.0)
		curCfg->Param_INT[parINT_NumZone].val[0] = 1.0;

	m->numZone = (INT)(curCfg->Param_INT[parINT_NumZone].val[0]);

	/////////////////////////////////////////////////////////////////////////
	if((curCalib->GenSetup[SETUP_MAPPING_ON]&MAPPING_SEGM))
		m->numZone = curCalib->GenSetup[SETUP_POLE_ELEMENTS] * 2;

	///////////////////////////////////////////////////////////////////////

}

DINT  DefaultCalibr_BPV_FACE_OSC(CurCalib_typ* defCalib){
UINT i;

		if(!defCalib)
			return 0;

		////////////////////////////////////////////////////////
		////   Default CALIBRATION

		i = CALIB_OSC_SFT_LIMIT;
		defCalib->Points[i].num = 4;

		defCalib->Points[i].val[0] = -1.0e+23;
		defCalib->Points[i].val[1] = 1.0e+23;
		defCalib->Points[i].val[2] = -1.0e+23;
		defCalib->Points[i].val[3] = 1.0e+23;

		i = CALIB_TIG_VOLT_FBK;
		defCalib->Points[i].num = 4;

		defCalib->Points[i].val[0] = 0.0; 	// 0 V
		defCalib->Points[i].val[1] = 1.44775391; 		// 6 V
		defCalib->Points[i].val[2] = 2.96142578; 		// 12 V
		defCalib->Points[i].val[3] = 4.45922852; 		// 18 V

		i = CALIB_TVL_SPEED_CMD;
		defCalib->Points[i].num = 8;

		// OMEGA 16 INCH  // 1"/min = 0.423 mm/s

		/*
		// Going Up
		defCalib->Points[i].val[0] = 0.846663; 	// X1 pos	 at 2"/min
		defCalib->Points[i].val[1] = 1.212983; 	// Y1 pos
		defCalib->Points[i].val[2] = 2.1166663; 	// X2 pos	at 5"/min
		defCalib->Points[i].val[3] = 2.621189; 	// Y2 pos

		// Going Down
		defCalib->Points[i].val[4] = 0.846663;		// X1 neg
		defCalib->Points[i].val[5] = 1.212983;		// Y1 neg
		defCalib->Points[i].val[6] = 2.1166663;	// X2 neg
		defCalib->Points[i].val[7] = 2.621189;	// Y2 neg
		*/

		defCalib->Points[i].val[0] = 0.0; 	// X1 pos	 at 2"/min
		defCalib->Points[i].val[1] = 0.0; 	// Y1 pos
		defCalib->Points[i].val[2] = 10.0; 	// X2 pos	at 5"/min
		defCalib->Points[i].val[3] = 10.0; 	// Y2 pos

		defCalib->Points[i].val[4] = 0.0;		// X1 neg
		defCalib->Points[i].val[5] = 0.0;		// Y1 neg
		defCalib->Points[i].val[6] = 10.0;	// X2 neg
		defCalib->Points[i].val[7] = 10.0;	// Y2 neg

		i = CALIB_WF_SPEED_CMD;
		defCalib->Points[i].num = 8;

		/*
		defCalib->Points[i].val[0] = 34.7; 	// X1 LEFT
		defCalib->Points[i].val[1] = 42.3; 	// Y1 LEFT
		defCalib->Points[i].val[2] = 70.6; 	// X2 LEFT
		defCalib->Points[i].val[3] = 84.7; 	// Y2 LEFT

		defCalib->Points[i].val[4] = 34.7;	// X1 RIGHT
		defCalib->Points[i].val[5] = 42.3;	// Y1 RIGHT
		defCalib->Points[i].val[6] = 70.6;	// X2 RIGHT
		defCalib->Points[i].val[7] = 84.7;	// Y2 RIGHT

		*/

		defCalib->Points[i].val[0] = 0.0; 	// X1 LEFT
		defCalib->Points[i].val[1] = 0.0; 	// Y1 LEFT
		defCalib->Points[i].val[2] = 10.0; 	// X2 LEFT
		defCalib->Points[i].val[3] = 10.0; 	// Y2 LEFT

		defCalib->Points[i].val[4] = 0.0;	// X1 RIGHT
		defCalib->Points[i].val[5] = 0.0;	// Y1 RIGHT
		defCalib->Points[i].val[6] = 10.0;	// X2 RIGHT
		defCalib->Points[i].val[7] = 10.0;	// Y2 RIGHT

		i = CALIB_WP_SPEED_CMD;
		defCalib->Points[i].num = 8;

		defCalib->Points[i].val[0] = 0.0;	// X1 LEFT
		defCalib->Points[i].val[1] = 0.0;	// Y1 LEFT
		defCalib->Points[i].val[2] = 10.0;	// X2 LEFT
		defCalib->Points[i].val[3] = 10.0;	// Y2 LEFT

		defCalib->Points[i].val[4] = 0.0;	// X1 RIGHT
		defCalib->Points[i].val[5] = 0.0;	// Y1 RIGHT
		defCalib->Points[i].val[6] = 10.0;	// X2 RIGHT
		defCalib->Points[i].val[7] = 10.0;	// Y2 RIGHT

		i=CALIB_TIG_AMPS_CMD;
		defCalib->Points[i].num = 4;
		/*
		defCalib->Points[i].val[0] = 92.0;	// X1
		defCalib->Points[i].val[1] = 80.0;	// Y1
		defCalib->Points[i].val[2] = 171.0; // X2
		defCalib->Points[i].val[3] = 150.0; // Y2
		defCalib->Points[i].num = 4;
		*/

		defCalib->Points[i].val[0] = 0.0; 	// X1
		defCalib->Points[i].val[1] = 0.0; 	// Y1
		defCalib->Points[i].val[2] = 500.0; // X2
		defCalib->Points[i].val[3] = 500.0; // Y2

		i=CALIB_HW_AMPS_CMD;
		defCalib->Points[i].num = 4;

		/*
		defCalib->Points[i].val[0] = 36.0;	// X1
		defCalib->Points[i].val[1] = 36.0;	// Y1
		defCalib->Points[i].val[2] = 83.0; // X2  - 160 amp max
		defCalib->Points[i].val[3] = 80.0; // Y2
		*/

		defCalib->Points[i].val[0] = 0.0;	// X1
		defCalib->Points[i].val[1] = 0.0;	// Y1
		defCalib->Points[i].val[2] = 80.0; // X2  - 160 amp max
		defCalib->Points[i].val[3] = 80.0; // Y2

		//// How many calibrations we have
		defCalib->num = 7;
		//////////////////////////////////////////////////////////////////////////////////

		return 1;

}

DINT  DefaultCalibr_BPV_v2_MT(CurCalib_typ* defCalib){
UINT i;

		if(!defCalib)
			return 0;

		////////////////////////////////////////////////////////
		////   Default CALIBRATION

		i = CALIB_OSC_SFT_LIMIT;
		defCalib->Points[i].num = 4;

		defCalib->Points[i].val[0] = -1.0e+23;
		defCalib->Points[i].val[1] = 1.0e+23;
		defCalib->Points[i].val[2] = -1.0e+23;
		defCalib->Points[i].val[3] = 1.0e+23;

		i = CALIB_TIG_VOLT_FBK;
		defCalib->Points[i].num = 4;

		defCalib->Points[i].val[0] = 0.377; 	// 0 V
		defCalib->Points[i].val[1] = 1.667; 	// 6 V
		defCalib->Points[i].val[2] = 3.08; 		// 12 V
		defCalib->Points[i].val[3] = 4.477; 	// 18 V

		i = CALIB_TVL_SPEED_CMD;
		defCalib->Points[i].num = 8;

		defCalib->Points[i].val[0] = 0.0; 	// X1 pos	 at 2"/min
		defCalib->Points[i].val[1] = 0.0; 	// Y1 pos
		defCalib->Points[i].val[2] = 10.0; 	// X2 pos	at 5"/min
		defCalib->Points[i].val[3] = 10.0; 	// Y2 pos

		defCalib->Points[i].val[4] = 0.0;		// X1 neg
		defCalib->Points[i].val[5] = 0.0;		// Y1 neg
		defCalib->Points[i].val[6] = 10.0;	// X2 neg
		defCalib->Points[i].val[7] = 10.0;	// Y2 neg

		i = CALIB_WF_SPEED_CMD;
		defCalib->Points[i].num = 8;

		defCalib->Points[i].val[0] = 0.0; 	// X1 LEFT
		defCalib->Points[i].val[1] = 0.0; 	// Y1 LEFT
		defCalib->Points[i].val[2] = 10.0; 	// X2 LEFT
		defCalib->Points[i].val[3] = 10.0; 	// Y2 LEFT

		defCalib->Points[i].val[4] = 0.0;	// X1 RIGHT
		defCalib->Points[i].val[5] = 0.0;	// Y1 RIGHT
		defCalib->Points[i].val[6] = 10.0;	// X2 RIGHT
		defCalib->Points[i].val[7] = 10.0;	// Y2 RIGHT

		i = CALIB_WP_SPEED_CMD;
		defCalib->Points[i].num = 8;

		defCalib->Points[i].val[0] = 0.0;	// X1 LEFT
		defCalib->Points[i].val[1] = 0.0;	// Y1 LEFT
		defCalib->Points[i].val[2] = 10.0;	// X2 LEFT
		defCalib->Points[i].val[3] = 10.0;	// Y2 LEFT

		defCalib->Points[i].val[4] = 0.0;	// X1 RIGHT
		defCalib->Points[i].val[5] = 0.0;	// Y1 RIGHT
		defCalib->Points[i].val[6] = 10.0;	// X2 RIGHT
		defCalib->Points[i].val[7] = 10.0;	// Y2 RIGHT

		i=CALIB_TIG_AMPS_CMD;
		defCalib->Points[i].num = 4;

		defCalib->Points[i].val[0] = 0.0; 	// X1
		defCalib->Points[i].val[1] = 0.0; 	// Y1
		defCalib->Points[i].val[2] = 500.0; // X2
		defCalib->Points[i].val[3] = 500.0; // Y2

		i=CALIB_HW_AMPS_CMD;
		defCalib->Points[i].num = 4;

		defCalib->Points[i].val[0] = 0.0;	// X1
		defCalib->Points[i].val[1] = 0.0;	// Y1
		defCalib->Points[i].val[2] = 80.0; // X2  - 160 amp max
		defCalib->Points[i].val[3] = 80.0; // Y2

		i=CALIB_INDX_CMD;
		defCalib->Points[i].num = 4;

		defCalib->Points[i].val[0] = 0.0; 	// X1
		defCalib->Points[i].val[1] = 0.0; 	// Y1
		defCalib->Points[i].val[2] = 500.0; // X2
		defCalib->Points[i].val[3] = 500.0; // Y2

		//// How many calibrations we have
		defCalib->num = 8;
		//////////////////////////////////////////////////////////////////////////////////

		return 1;

}
DINT  DefaultCalibr_BPV_v2(CurCalib_typ* defCalib){
UINT i;

		if(!defCalib)
			return 0;

		////////////////////////////////////////////////////////
		////   Default CALIBRATION

		i = CALIB_OSC_SFT_LIMIT;
		defCalib->Points[i].num = 4;

		defCalib->Points[i].val[0] = -1.0e+23;
		defCalib->Points[i].val[1] = 1.0e+23;
		defCalib->Points[i].val[2] = -1.0e+23;
		defCalib->Points[i].val[3] = 1.0e+23;

		i = CALIB_TIG_VOLT_FBK;
		defCalib->Points[i].num = 4;

		defCalib->Points[i].val[0] = 0.377; 	// 0 V
		defCalib->Points[i].val[1] = 1.667; 	// 6 V
		defCalib->Points[i].val[2] = 3.08; 		// 12 V
		defCalib->Points[i].val[3] = 4.477; 	// 18 V

		i = CALIB_TVL_SPEED_CMD;
		defCalib->Points[i].num = 8;

		defCalib->Points[i].val[0] = 0.0; 	// X1 pos	 at 2"/min
		defCalib->Points[i].val[1] = 0.0; 	// Y1 pos
		defCalib->Points[i].val[2] = 10.0; 	// X2 pos	at 5"/min
		defCalib->Points[i].val[3] = 10.0; 	// Y2 pos

		defCalib->Points[i].val[4] = 0.0;		// X1 neg
		defCalib->Points[i].val[5] = 0.0;		// Y1 neg
		defCalib->Points[i].val[6] = 10.0;	// X2 neg
		defCalib->Points[i].val[7] = 10.0;	// Y2 neg

		i = CALIB_WF_SPEED_CMD;
		defCalib->Points[i].num = 8;

		defCalib->Points[i].val[0] = 0.0; 	// X1 LEFT
		defCalib->Points[i].val[1] = 0.0; 	// Y1 LEFT
		defCalib->Points[i].val[2] = 10.0; 	// X2 LEFT
		defCalib->Points[i].val[3] = 10.0; 	// Y2 LEFT

		defCalib->Points[i].val[4] = 0.0;	// X1 RIGHT
		defCalib->Points[i].val[5] = 0.0;	// Y1 RIGHT
		defCalib->Points[i].val[6] = 10.0;	// X2 RIGHT
		defCalib->Points[i].val[7] = 10.0;	// Y2 RIGHT

		i = CALIB_WP_SPEED_CMD;
		defCalib->Points[i].num = 8;

		defCalib->Points[i].val[0] = 0.0;	// X1 LEFT
		defCalib->Points[i].val[1] = 0.0;	// Y1 LEFT
		defCalib->Points[i].val[2] = 10.0;	// X2 LEFT
		defCalib->Points[i].val[3] = 10.0;	// Y2 LEFT

		defCalib->Points[i].val[4] = 0.0;	// X1 RIGHT
		defCalib->Points[i].val[5] = 0.0;	// Y1 RIGHT
		defCalib->Points[i].val[6] = 10.0;	// X2 RIGHT
		defCalib->Points[i].val[7] = 10.0;	// Y2 RIGHT

		i=CALIB_TIG_AMPS_CMD;
		defCalib->Points[i].num = 4;

		defCalib->Points[i].val[0] = 0.0; 	// X1
		defCalib->Points[i].val[1] = 0.0; 	// Y1
		defCalib->Points[i].val[2] = 500.0; // X2
		defCalib->Points[i].val[3] = 500.0; // Y2

		i=CALIB_HW_AMPS_CMD;
		defCalib->Points[i].num = 4;

		defCalib->Points[i].val[0] = 0.0;	// X1
		defCalib->Points[i].val[1] = 0.0;	// Y1
		defCalib->Points[i].val[2] = 80.0; // X2  - 160 amp max
		defCalib->Points[i].val[3] = 80.0; // Y2

		i=CALIB_INDX_CMD;
		defCalib->Points[i].num = 4;

		defCalib->Points[i].val[0] = 0.0; 	// X1
		defCalib->Points[i].val[1] = 0.0; 	// Y1
		defCalib->Points[i].val[2] = 500.0; // X2
		defCalib->Points[i].val[3] = 500.0; // Y2

		//// How many calibrations we have
		defCalib->num = 8;
		//////////////////////////////////////////////////////////////////////////////////

		return 1;

}

DINT  DefaultCalibr_MIG_TIG(CurCalib_typ* defCalib){
UINT i;

		if(!defCalib)
			return 0;

		////////////////////////////////////////////////////////
		////   Default CALIBRATION

		i = CALIB_OSC_SFT_LIMIT;
		defCalib->Points[i].num = 4;

		defCalib->Points[i].val[0] = -1.0e+23;
		defCalib->Points[i].val[1] = 1.0e+23;
		defCalib->Points[i].val[2] = -1.0e+23;
		defCalib->Points[i].val[3] = 1.0e+23;

		i = CALIB_TIG_VOLT_FBK;
		defCalib->Points[i].num = 4;

		defCalib->Points[i].val[0] = 0.377; 	// 0 V
		defCalib->Points[i].val[1] = 1.667; 	// 6 V
		defCalib->Points[i].val[2] = 3.08; 		// 12 V
		defCalib->Points[i].val[3] = 4.477; 	// 18 V

		i = CALIB_TVL_SPEED_CMD;
		defCalib->Points[i].num = 8;

		defCalib->Points[i].val[0] = 0.0; 	// X1 pos	 at 2"/min
		defCalib->Points[i].val[1] = 0.0; 	// Y1 pos
		defCalib->Points[i].val[2] = 10.0; 	// X2 pos	at 5"/min
		defCalib->Points[i].val[3] = 10.0; 	// Y2 pos

		defCalib->Points[i].val[4] = 0.0;		// X1 neg
		defCalib->Points[i].val[5] = 0.0;		// Y1 neg
		defCalib->Points[i].val[6] = 10.0;	// X2 neg
		defCalib->Points[i].val[7] = 10.0;	// Y2 neg

		i = CALIB_WF_SPEED_CMD;
		defCalib->Points[i].num = 8;

		defCalib->Points[i].val[0] = 0.0; 	// X1 LEFT
		defCalib->Points[i].val[1] = 0.0; 	// Y1 LEFT
		defCalib->Points[i].val[2] = 10.0; 	// X2 LEFT
		defCalib->Points[i].val[3] = 10.0; 	// Y2 LEFT

		defCalib->Points[i].val[4] = 0.0;	// X1 RIGHT
		defCalib->Points[i].val[5] = 0.0;	// Y1 RIGHT
		defCalib->Points[i].val[6] = 10.0;	// X2 RIGHT
		defCalib->Points[i].val[7] = 10.0;	// Y2 RIGHT

		i = CALIB_WP_SPEED_CMD;
		defCalib->Points[i].num = 8;

		defCalib->Points[i].val[0] = 0.0;	// X1 LEFT
		defCalib->Points[i].val[1] = 0.0;	// Y1 LEFT
		defCalib->Points[i].val[2] = 10.0;	// X2 LEFT
		defCalib->Points[i].val[3] = 10.0;	// Y2 LEFT

		defCalib->Points[i].val[4] = 0.0;	// X1 RIGHT
		defCalib->Points[i].val[5] = 0.0;	// Y1 RIGHT
		defCalib->Points[i].val[6] = 10.0;	// X2 RIGHT
		defCalib->Points[i].val[7] = 10.0;	// Y2 RIGHT

		i=CALIB_TIG_AMPS_CMD;
		defCalib->Points[i].num = 4;

		defCalib->Points[i].val[0] = 0.0; 	// X1
		defCalib->Points[i].val[1] = 0.0; 	// Y1
		defCalib->Points[i].val[2] = 500.0; // X2
		defCalib->Points[i].val[3] = 500.0; // Y2

		i=CALIB_HW_AMPS_CMD;
		defCalib->Points[i].num = 4;

		defCalib->Points[i].val[0] = 0.0;	// X1
		defCalib->Points[i].val[1] = 0.0;	// Y1
		defCalib->Points[i].val[2] = 80.0; // X2  - 160 amp max
		defCalib->Points[i].val[3] = 80.0; // Y2

		i=CALIB_INDX_CMD;
		defCalib->Points[i].num = 4;

		defCalib->Points[i].val[0] = 0.0; 	// X1
		defCalib->Points[i].val[1] = 0.0; 	// Y1
		defCalib->Points[i].val[2] = 500.0; // X2
		defCalib->Points[i].val[3] = 500.0; // Y2

		//// How many calibrations we have
		defCalib->num = 8;
		//////////////////////////////////////////////////////////////////////////////////

		return 1;

}
///////////////////////////////////////////////////////////////

DINT  DefaultCalibr_BPV_v2_MT_BO(CurCalib_typ* defCalib){
UINT i;

		if(!defCalib)
			return 0;

		////////////////////////////////////////////////////////
		////   Default CALIBRATION

		i = CALIB_OSC_SFT_LIMIT;
		defCalib->Points[i].num = 4;

		defCalib->Points[i].val[0] = -1.0e+23;
		defCalib->Points[i].val[1] = 1.0e+23;
		defCalib->Points[i].val[2] = -1.0e+23;
		defCalib->Points[i].val[3] = 1.0e+23;

		i = CALIB_TIG_VOLT_FBK;
		defCalib->Points[i].num = 4;

		defCalib->Points[i].val[0] = 0.377; 	// 0 V
		defCalib->Points[i].val[1] = 1.667; 	// 6 V
		defCalib->Points[i].val[2] = 3.08; 		// 12 V
		defCalib->Points[i].val[3] = 4.477; 	// 18 V

		i = CALIB_TVL_SPEED_CMD;
		defCalib->Points[i].num = 8;

		defCalib->Points[i].val[0] = 0.0; 	// X1 pos	 at 2"/min
		defCalib->Points[i].val[1] = 0.0; 	// Y1 pos
		defCalib->Points[i].val[2] = 10.0; 	// X2 pos	at 5"/min
		defCalib->Points[i].val[3] = 10.0; 	// Y2 pos

		defCalib->Points[i].val[4] = 0.0;		// X1 neg
		defCalib->Points[i].val[5] = 0.0;		// Y1 neg
		defCalib->Points[i].val[6] = 10.0;	// X2 neg
		defCalib->Points[i].val[7] = 10.0;	// Y2 neg

		i = CALIB_WF_SPEED_CMD;
		defCalib->Points[i].num = 8;

		defCalib->Points[i].val[0] = 0.0; 	// X1 LEFT
		defCalib->Points[i].val[1] = 0.0; 	// Y1 LEFT
		defCalib->Points[i].val[2] = 10.0; 	// X2 LEFT
		defCalib->Points[i].val[3] = 10.0; 	// Y2 LEFT

		defCalib->Points[i].val[4] = 0.0;	// X1 RIGHT
		defCalib->Points[i].val[5] = 0.0;	// Y1 RIGHT
		defCalib->Points[i].val[6] = 10.0;	// X2 RIGHT
		defCalib->Points[i].val[7] = 10.0;	// Y2 RIGHT

		i = CALIB_WP_SPEED_CMD;
		defCalib->Points[i].num = 8;

		defCalib->Points[i].val[0] = 0.0;	// X1 LEFT
		defCalib->Points[i].val[1] = 0.0;	// Y1 LEFT
		defCalib->Points[i].val[2] = 10.0;	// X2 LEFT
		defCalib->Points[i].val[3] = 10.0;	// Y2 LEFT

		defCalib->Points[i].val[4] = 0.0;	// X1 RIGHT
		defCalib->Points[i].val[5] = 0.0;	// Y1 RIGHT
		defCalib->Points[i].val[6] = 10.0;	// X2 RIGHT
		defCalib->Points[i].val[7] = 10.0;	// Y2 RIGHT

		i=CALIB_TIG_AMPS_CMD;
		defCalib->Points[i].num = 4;

		defCalib->Points[i].val[0] = 0.0; 	// X1
		defCalib->Points[i].val[1] = 0.0; 	// Y1
		defCalib->Points[i].val[2] = 500.0; // X2
		defCalib->Points[i].val[3] = 500.0; // Y2

		i=CALIB_HW_AMPS_CMD;
		defCalib->Points[i].num = 4;

		defCalib->Points[i].val[0] = 0.0;	// X1
		defCalib->Points[i].val[1] = 0.0;	// Y1
		defCalib->Points[i].val[2] = 80.0; // X2  - 160 amp max
		defCalib->Points[i].val[3] = 80.0; // Y2

		i=CALIB_INDX_CMD;
		defCalib->Points[i].num = 4;

		defCalib->Points[i].val[0] = 0.0; 	// X1
		defCalib->Points[i].val[1] = 0.0; 	// Y1
		defCalib->Points[i].val[2] = 500.0; // X2
		defCalib->Points[i].val[3] = 500.0; // Y2

		//// How many calibrations we have
		defCalib->num = 8;
		//////////////////////////////////////////////////////////////////////////////////

		return 1;

}

DINT  DefaultCalibr_BPV_v2_TT_BO(CurCalib_typ* defCalib){
UINT i;

		if(!defCalib)
			return 0;

		////////////////////////////////////////////////////////
		////   Default CALIBRATION

		i = CALIB_OSC_SFT_LIMIT;
		defCalib->Points[i].num = 4;

		defCalib->Points[i].val[0] = -1.0e+23;
		defCalib->Points[i].val[1] = 1.0e+23;
		defCalib->Points[i].val[2] = -1.0e+23;
		defCalib->Points[i].val[3] = 1.0e+23;

		i = CALIB_TIG_VOLT_FBK;
		defCalib->Points[i].num = 4;

		defCalib->Points[i].val[0] = 0.377; 	// 0 V
		defCalib->Points[i].val[1] = 1.667; 	// 6 V
		defCalib->Points[i].val[2] = 3.08; 		// 12 V
		defCalib->Points[i].val[3] = 4.477; 	// 18 V

		i = CALIB_TVL_SPEED_CMD;
		defCalib->Points[i].num = 8;

		defCalib->Points[i].val[0] = 0.0; 	// X1 pos	 at 2"/min
		defCalib->Points[i].val[1] = 0.0; 	// Y1 pos
		defCalib->Points[i].val[2] = 10.0; 	// X2 pos	at 5"/min
		defCalib->Points[i].val[3] = 10.0; 	// Y2 pos

		defCalib->Points[i].val[4] = 0.0;		// X1 neg
		defCalib->Points[i].val[5] = 0.0;		// Y1 neg
		defCalib->Points[i].val[6] = 10.0;	// X2 neg
		defCalib->Points[i].val[7] = 10.0;	// Y2 neg

		i = CALIB_WF_SPEED_CMD;
		defCalib->Points[i].num = 8;

		defCalib->Points[i].val[0] = 0.0; 	// X1 LEFT
		defCalib->Points[i].val[1] = 0.0; 	// Y1 LEFT
		defCalib->Points[i].val[2] = 10.0; 	// X2 LEFT
		defCalib->Points[i].val[3] = 10.0; 	// Y2 LEFT

		defCalib->Points[i].val[4] = 0.0;	// X1 RIGHT
		defCalib->Points[i].val[5] = 0.0;	// Y1 RIGHT
		defCalib->Points[i].val[6] = 10.0;	// X2 RIGHT
		defCalib->Points[i].val[7] = 10.0;	// Y2 RIGHT

		i = CALIB_WP_SPEED_CMD;
		defCalib->Points[i].num = 8;

		defCalib->Points[i].val[0] = 0.0;	// X1 LEFT
		defCalib->Points[i].val[1] = 0.0;	// Y1 LEFT
		defCalib->Points[i].val[2] = 10.0;	// X2 LEFT
		defCalib->Points[i].val[3] = 10.0;	// Y2 LEFT

		defCalib->Points[i].val[4] = 0.0;	// X1 RIGHT
		defCalib->Points[i].val[5] = 0.0;	// Y1 RIGHT
		defCalib->Points[i].val[6] = 10.0;	// X2 RIGHT
		defCalib->Points[i].val[7] = 10.0;	// Y2 RIGHT

		i=CALIB_TIG_AMPS_CMD;
		defCalib->Points[i].num = 4;

		defCalib->Points[i].val[0] = 0.0; 	// X1
		defCalib->Points[i].val[1] = 0.0; 	// Y1
		defCalib->Points[i].val[2] = 500.0; // X2
		defCalib->Points[i].val[3] = 500.0; // Y2

		i=CALIB_HW_AMPS_CMD;
		defCalib->Points[i].num = 4;

		defCalib->Points[i].val[0] = 0.0;	// X1
		defCalib->Points[i].val[1] = 0.0;	// Y1
		defCalib->Points[i].val[2] = 80.0; // X2  - 160 amp max
		defCalib->Points[i].val[3] = 80.0; // Y2

		i=CALIB_INDX_CMD;
		defCalib->Points[i].num = 4;

		defCalib->Points[i].val[0] = 0.0; 	// X1
		defCalib->Points[i].val[1] = 0.0; 	// Y1
		defCalib->Points[i].val[2] = 500.0; // X2
		defCalib->Points[i].val[3] = 500.0; // Y2

		//// How many calibrations we have
		defCalib->num = 8;
		//////////////////////////////////////////////////////////////////////////////////

		return 1;

}
DINT  DefaultCalibr_BPV_v2_MT_BO_TOS(CurCalib_typ* defCalib){
UINT i;

		if(!defCalib)
			return 0;

		////////////////////////////////////////////////////////
		////   Default CALIBRATION

		i = CALIB_OSC_SFT_LIMIT;
		defCalib->Points[i].num = 4;

		defCalib->Points[i].val[0] = -1.0e+23;
		defCalib->Points[i].val[1] = 1.0e+23;
		defCalib->Points[i].val[2] = -1.0e+23;
		defCalib->Points[i].val[3] = 1.0e+23;

		i = CALIB_TIG_VOLT_FBK;
		defCalib->Points[i].num = 4;

		defCalib->Points[i].val[0] = 0.377; 	// 0 V
		defCalib->Points[i].val[1] = 1.667; 	// 6 V
		defCalib->Points[i].val[2] = 3.08; 		// 12 V
		defCalib->Points[i].val[3] = 4.477; 	// 18 V

		i = CALIB_TVL_SPEED_CMD;
		defCalib->Points[i].num = 8;

		defCalib->Points[i].val[0] = 0.0; 	// X1 pos	 at 2"/min
		defCalib->Points[i].val[1] = 0.0; 	// Y1 pos
		defCalib->Points[i].val[2] = 10.0; 	// X2 pos	at 5"/min
		defCalib->Points[i].val[3] = 10.0; 	// Y2 pos

		defCalib->Points[i].val[4] = 0.0;		// X1 neg
		defCalib->Points[i].val[5] = 0.0;		// Y1 neg
		defCalib->Points[i].val[6] = 10.0;	// X2 neg
		defCalib->Points[i].val[7] = 10.0;	// Y2 neg

		i = CALIB_WF_SPEED_CMD;
		defCalib->Points[i].num = 8;

		defCalib->Points[i].val[0] = 0.0; 	// X1 LEFT
		defCalib->Points[i].val[1] = 0.0; 	// Y1 LEFT
		defCalib->Points[i].val[2] = 10.0; 	// X2 LEFT
		defCalib->Points[i].val[3] = 10.0; 	// Y2 LEFT

		defCalib->Points[i].val[4] = 0.0;	// X1 RIGHT
		defCalib->Points[i].val[5] = 0.0;	// Y1 RIGHT
		defCalib->Points[i].val[6] = 10.0;	// X2 RIGHT
		defCalib->Points[i].val[7] = 10.0;	// Y2 RIGHT

		i = CALIB_WP_SPEED_CMD;
		defCalib->Points[i].num = 8;

		defCalib->Points[i].val[0] = 0.0;	// X1 LEFT
		defCalib->Points[i].val[1] = 0.0;	// Y1 LEFT
		defCalib->Points[i].val[2] = 10.0;	// X2 LEFT
		defCalib->Points[i].val[3] = 10.0;	// Y2 LEFT

		defCalib->Points[i].val[4] = 0.0;	// X1 RIGHT
		defCalib->Points[i].val[5] = 0.0;	// Y1 RIGHT
		defCalib->Points[i].val[6] = 10.0;	// X2 RIGHT
		defCalib->Points[i].val[7] = 10.0;	// Y2 RIGHT

		i=CALIB_TIG_AMPS_CMD;
		defCalib->Points[i].num = 4;

		defCalib->Points[i].val[0] = 0.0; 	// X1
		defCalib->Points[i].val[1] = 0.0; 	// Y1
		defCalib->Points[i].val[2] = 500.0; // X2
		defCalib->Points[i].val[3] = 500.0; // Y2

		i=CALIB_HW_AMPS_CMD;
		defCalib->Points[i].num = 4;

		defCalib->Points[i].val[0] = 0.0;	// X1
		defCalib->Points[i].val[1] = 0.0;	// Y1
		defCalib->Points[i].val[2] = 80.0; // X2  - 160 amp max
		defCalib->Points[i].val[3] = 80.0; // Y2

		i=CALIB_INDX_CMD;
		defCalib->Points[i].num = 4;

		defCalib->Points[i].val[0] = 0.0; 	// X1
		defCalib->Points[i].val[1] = 0.0; 	// Y1
		defCalib->Points[i].val[2] = 500.0; // X2
		defCalib->Points[i].val[3] = 500.0; // Y2

		//// How many calibrations we have
		defCalib->num = 8;
		//////////////////////////////////////////////////////////////////////////////////

		return 1;

}
DINT  DefaultCalibr_BPV_v2_TT_BO_TOS(CurCalib_typ* defCalib){
UINT i;

		if(!defCalib)
			return 0;

		////////////////////////////////////////////////////////
		////   Default CALIBRATION

		i = CALIB_OSC_SFT_LIMIT;
		defCalib->Points[i].num = 4;

		defCalib->Points[i].val[0] = -1.0e+23;
		defCalib->Points[i].val[1] = 1.0e+23;
		defCalib->Points[i].val[2] = -1.0e+23;
		defCalib->Points[i].val[3] = 1.0e+23;

		i = CALIB_TIG_VOLT_FBK;
		defCalib->Points[i].num = 4;

		defCalib->Points[i].val[0] = 0.377; 	// 0 V
		defCalib->Points[i].val[1] = 1.667; 	// 6 V
		defCalib->Points[i].val[2] = 3.08; 		// 12 V
		defCalib->Points[i].val[3] = 4.477; 	// 18 V

		i = CALIB_TVL_SPEED_CMD;
		defCalib->Points[i].num = 8;

		defCalib->Points[i].val[0] = 0.0; 	// X1 pos	 at 2"/min
		defCalib->Points[i].val[1] = 0.0; 	// Y1 pos
		defCalib->Points[i].val[2] = 10.0; 	// X2 pos	at 5"/min
		defCalib->Points[i].val[3] = 10.0; 	// Y2 pos

		defCalib->Points[i].val[4] = 0.0;		// X1 neg
		defCalib->Points[i].val[5] = 0.0;		// Y1 neg
		defCalib->Points[i].val[6] = 10.0;	// X2 neg
		defCalib->Points[i].val[7] = 10.0;	// Y2 neg

		i = CALIB_WF_SPEED_CMD;
		defCalib->Points[i].num = 8;

		defCalib->Points[i].val[0] = 0.0; 	// X1 LEFT
		defCalib->Points[i].val[1] = 0.0; 	// Y1 LEFT
		defCalib->Points[i].val[2] = 10.0; 	// X2 LEFT
		defCalib->Points[i].val[3] = 10.0; 	// Y2 LEFT

		defCalib->Points[i].val[4] = 0.0;	// X1 RIGHT
		defCalib->Points[i].val[5] = 0.0;	// Y1 RIGHT
		defCalib->Points[i].val[6] = 10.0;	// X2 RIGHT
		defCalib->Points[i].val[7] = 10.0;	// Y2 RIGHT

		i = CALIB_WP_SPEED_CMD;
		defCalib->Points[i].num = 8;

		defCalib->Points[i].val[0] = 0.0;	// X1 LEFT
		defCalib->Points[i].val[1] = 0.0;	// Y1 LEFT
		defCalib->Points[i].val[2] = 10.0;	// X2 LEFT
		defCalib->Points[i].val[3] = 10.0;	// Y2 LEFT

		defCalib->Points[i].val[4] = 0.0;	// X1 RIGHT
		defCalib->Points[i].val[5] = 0.0;	// Y1 RIGHT
		defCalib->Points[i].val[6] = 10.0;	// X2 RIGHT
		defCalib->Points[i].val[7] = 10.0;	// Y2 RIGHT

		i=CALIB_TIG_AMPS_CMD;
		defCalib->Points[i].num = 4;

		defCalib->Points[i].val[0] = 0.0; 	// X1
		defCalib->Points[i].val[1] = 0.0; 	// Y1
		defCalib->Points[i].val[2] = 500.0; // X2
		defCalib->Points[i].val[3] = 500.0; // Y2

		i=CALIB_HW_AMPS_CMD;
		defCalib->Points[i].num = 4;

		defCalib->Points[i].val[0] = 0.0;	// X1
		defCalib->Points[i].val[1] = 0.0;	// Y1
		defCalib->Points[i].val[2] = 80.0; // X2  - 160 amp max
		defCalib->Points[i].val[3] = 80.0; // Y2

		i=CALIB_INDX_CMD;
		defCalib->Points[i].num = 4;

		defCalib->Points[i].val[0] = 0.0; 	// X1
		defCalib->Points[i].val[1] = 0.0; 	// Y1
		defCalib->Points[i].val[2] = 500.0; // X2
		defCalib->Points[i].val[3] = 500.0; // Y2

		//// How many calibrations we have
		defCalib->num = 8;
		//////////////////////////////////////////////////////////////////////////////////

		return 1;

}

DINT  DefaultCalibr_BPV_v2_MPBO(CurCalib_typ* defCalib){
UINT i;

		if(!defCalib)
			return 0;

		////////////////////////////////////////////////////////
		////   Default CALIBRATION

		i = CALIB_OSC_SFT_LIMIT;
		defCalib->Points[i].num = 4;

		defCalib->Points[i].val[0] = -1.0e+23;
		defCalib->Points[i].val[1] = 1.0e+23;
		defCalib->Points[i].val[2] = -1.0e+23;
		defCalib->Points[i].val[3] = 1.0e+23;

		i = CALIB_TIG_VOLT_FBK;
		defCalib->Points[i].num = 4;

		defCalib->Points[i].val[0] = 0.377; 	// 0 V
		defCalib->Points[i].val[1] = 1.667; 	// 6 V
		defCalib->Points[i].val[2] = 3.08; 		// 12 V
		defCalib->Points[i].val[3] = 4.477; 	// 18 V

		i = CALIB_TVL_SPEED_CMD;
		defCalib->Points[i].num = 8;

		defCalib->Points[i].val[0] = 0.0; 	// X1 pos	 at 2"/min
		defCalib->Points[i].val[1] = 0.0; 	// Y1 pos
		defCalib->Points[i].val[2] = 10.0; 	// X2 pos	at 5"/min
		defCalib->Points[i].val[3] = 10.0; 	// Y2 pos

		defCalib->Points[i].val[4] = 0.0;		// X1 neg
		defCalib->Points[i].val[5] = 0.0;		// Y1 neg
		defCalib->Points[i].val[6] = 10.0;	// X2 neg
		defCalib->Points[i].val[7] = 10.0;	// Y2 neg

		i = CALIB_WF_SPEED_CMD;
		defCalib->Points[i].num = 8;

		defCalib->Points[i].val[0] = 0.0; 	// X1 LEFT
		defCalib->Points[i].val[1] = 0.0; 	// Y1 LEFT
		defCalib->Points[i].val[2] = 10.0; 	// X2 LEFT
		defCalib->Points[i].val[3] = 10.0; 	// Y2 LEFT

		defCalib->Points[i].val[4] = 0.0;	// X1 RIGHT
		defCalib->Points[i].val[5] = 0.0;	// Y1 RIGHT
		defCalib->Points[i].val[6] = 10.0;	// X2 RIGHT
		defCalib->Points[i].val[7] = 10.0;	// Y2 RIGHT

		i = CALIB_WP_SPEED_CMD;
		defCalib->Points[i].num = 8;

		defCalib->Points[i].val[0] = 0.0;	// X1 LEFT
		defCalib->Points[i].val[1] = 0.0;	// Y1 LEFT
		defCalib->Points[i].val[2] = 10.0;	// X2 LEFT
		defCalib->Points[i].val[3] = 10.0;	// Y2 LEFT

		defCalib->Points[i].val[4] = 0.0;	// X1 RIGHT
		defCalib->Points[i].val[5] = 0.0;	// Y1 RIGHT
		defCalib->Points[i].val[6] = 10.0;	// X2 RIGHT
		defCalib->Points[i].val[7] = 10.0;	// Y2 RIGHT

		i=CALIB_TIG_AMPS_CMD;
		defCalib->Points[i].num = 4;

		defCalib->Points[i].val[0] = 0.0; 	// X1
		defCalib->Points[i].val[1] = 0.0; 	// Y1
		defCalib->Points[i].val[2] = 500.0; // X2
		defCalib->Points[i].val[3] = 500.0; // Y2

		i=CALIB_HW_AMPS_CMD;
		defCalib->Points[i].num = 4;

		defCalib->Points[i].val[0] = 0.0;	// X1
		defCalib->Points[i].val[1] = 0.0;	// Y1
		defCalib->Points[i].val[2] = 80.0; // X2  - 160 amp max
		defCalib->Points[i].val[3] = 80.0; // Y2

		i=CALIB_INDX_CMD;
		defCalib->Points[i].num = 4;

		defCalib->Points[i].val[0] = 0.0; 	// X1
		defCalib->Points[i].val[1] = 0.0; 	// Y1
		defCalib->Points[i].val[2] = 500.0; // X2
		defCalib->Points[i].val[3] = 500.0; // Y2

		//// How many calibrations we have
		defCalib->num = 8;
		//////////////////////////////////////////////////////////////////////////////////

		return 1;

}

DINT  DefaultCalibr_BPV_v2_MPGH(CurCalib_typ* defCalib){
UINT i;

		if(!defCalib)
			return 0;

		////////////////////////////////////////////////////////
		////   Default CALIBRATION

		i = CALIB_OSC_SFT_LIMIT;
		defCalib->Points[i].num = 4;

		defCalib->Points[i].val[0] = -1.0e+23;
		defCalib->Points[i].val[1] = 1.0e+23;
		defCalib->Points[i].val[2] = -1.0e+23;
		defCalib->Points[i].val[3] = 1.0e+23;

		i = CALIB_TIG_VOLT_FBK;
		defCalib->Points[i].num = 4;

		defCalib->Points[i].val[0] = 0.377; 	// 0 V
		defCalib->Points[i].val[1] = 1.667; 	// 6 V
		defCalib->Points[i].val[2] = 3.08; 		// 12 V
		defCalib->Points[i].val[3] = 4.477; 	// 18 V

		i = CALIB_TVL_SPEED_CMD;
		defCalib->Points[i].num = 8;

		defCalib->Points[i].val[0] = 0.0; 	// X1 pos	 at 2"/min
		defCalib->Points[i].val[1] = 0.0; 	// Y1 pos
		defCalib->Points[i].val[2] = 10.0; 	// X2 pos	at 5"/min
		defCalib->Points[i].val[3] = 10.0; 	// Y2 pos

		defCalib->Points[i].val[4] = 0.0;		// X1 neg
		defCalib->Points[i].val[5] = 0.0;		// Y1 neg
		defCalib->Points[i].val[6] = 10.0;	// X2 neg
		defCalib->Points[i].val[7] = 10.0;	// Y2 neg

		i = CALIB_WF_SPEED_CMD;
		defCalib->Points[i].num = 8;

		defCalib->Points[i].val[0] = 0.0; 	// X1 LEFT
		defCalib->Points[i].val[1] = 0.0; 	// Y1 LEFT
		defCalib->Points[i].val[2] = 10.0; 	// X2 LEFT
		defCalib->Points[i].val[3] = 10.0; 	// Y2 LEFT

		defCalib->Points[i].val[4] = 0.0;	// X1 RIGHT
		defCalib->Points[i].val[5] = 0.0;	// Y1 RIGHT
		defCalib->Points[i].val[6] = 10.0;	// X2 RIGHT
		defCalib->Points[i].val[7] = 10.0;	// Y2 RIGHT

		i = CALIB_WP_SPEED_CMD;
		defCalib->Points[i].num = 8;

		defCalib->Points[i].val[0] = 0.0;	// X1 LEFT
		defCalib->Points[i].val[1] = 0.0;	// Y1 LEFT
		defCalib->Points[i].val[2] = 10.0;	// X2 LEFT
		defCalib->Points[i].val[3] = 10.0;	// Y2 LEFT

		defCalib->Points[i].val[4] = 0.0;	// X1 RIGHT
		defCalib->Points[i].val[5] = 0.0;	// Y1 RIGHT
		defCalib->Points[i].val[6] = 10.0;	// X2 RIGHT
		defCalib->Points[i].val[7] = 10.0;	// Y2 RIGHT

		i=CALIB_TIG_AMPS_CMD;
		defCalib->Points[i].num = 4;

		defCalib->Points[i].val[0] = 0.0; 	// X1
		defCalib->Points[i].val[1] = 0.0; 	// Y1
		defCalib->Points[i].val[2] = 500.0; // X2
		defCalib->Points[i].val[3] = 500.0; // Y2

		i=CALIB_HW_AMPS_CMD;
		defCalib->Points[i].num = 4;

		defCalib->Points[i].val[0] = 0.0;	// X1
		defCalib->Points[i].val[1] = 0.0;	// Y1
		defCalib->Points[i].val[2] = 80.0; // X2  - 160 amp max
		defCalib->Points[i].val[3] = 80.0; // Y2

		i=CALIB_INDX_CMD;
		defCalib->Points[i].num = 4;

		defCalib->Points[i].val[0] = 0.0; 	// X1
		defCalib->Points[i].val[1] = 0.0; 	// Y1
		defCalib->Points[i].val[2] = 500.0; // X2
		defCalib->Points[i].val[3] = 500.0; // Y2

		//// How many calibrations we have
		defCalib->num = 8;
		//////////////////////////////////////////////////////////////////////////////////

		return 1;

}

DINT  DefaultCalibr_BPV_v2_MPGV(CurCalib_typ* defCalib){
UINT i;

		if(!defCalib)
			return 0;

		////////////////////////////////////////////////////////
		////   Default CALIBRATION

		i = CALIB_OSC_SFT_LIMIT;
		defCalib->Points[i].num = 4;

		defCalib->Points[i].val[0] = -1.0e+23;
		defCalib->Points[i].val[1] = 1.0e+23;
		defCalib->Points[i].val[2] = -1.0e+23;
		defCalib->Points[i].val[3] = 1.0e+23;

		i = CALIB_TIG_VOLT_FBK;
		defCalib->Points[i].num = 4;

		defCalib->Points[i].val[0] = 0.377; 	// 0 V
		defCalib->Points[i].val[1] = 1.667; 	// 6 V
		defCalib->Points[i].val[2] = 3.08; 		// 12 V
		defCalib->Points[i].val[3] = 4.477; 	// 18 V

		i = CALIB_TVL_SPEED_CMD;
		defCalib->Points[i].num = 8;

		defCalib->Points[i].val[0] = 0.0; 	// X1 pos	 at 2"/min
		defCalib->Points[i].val[1] = 0.0; 	// Y1 pos
		defCalib->Points[i].val[2] = 10.0; 	// X2 pos	at 5"/min
		defCalib->Points[i].val[3] = 10.0; 	// Y2 pos

		defCalib->Points[i].val[4] = 0.0;		// X1 neg
		defCalib->Points[i].val[5] = 0.0;		// Y1 neg
		defCalib->Points[i].val[6] = 10.0;	// X2 neg
		defCalib->Points[i].val[7] = 10.0;	// Y2 neg

		i = CALIB_WF_SPEED_CMD;
		defCalib->Points[i].num = 8;

		defCalib->Points[i].val[0] = 0.0; 	// X1 LEFT
		defCalib->Points[i].val[1] = 0.0; 	// Y1 LEFT
		defCalib->Points[i].val[2] = 10.0; 	// X2 LEFT
		defCalib->Points[i].val[3] = 10.0; 	// Y2 LEFT

		defCalib->Points[i].val[4] = 0.0;	// X1 RIGHT
		defCalib->Points[i].val[5] = 0.0;	// Y1 RIGHT
		defCalib->Points[i].val[6] = 10.0;	// X2 RIGHT
		defCalib->Points[i].val[7] = 10.0;	// Y2 RIGHT

		i = CALIB_WP_SPEED_CMD;
		defCalib->Points[i].num = 8;

		defCalib->Points[i].val[0] = 0.0;	// X1 LEFT
		defCalib->Points[i].val[1] = 0.0;	// Y1 LEFT
		defCalib->Points[i].val[2] = 10.0;	// X2 LEFT
		defCalib->Points[i].val[3] = 10.0;	// Y2 LEFT

		defCalib->Points[i].val[4] = 0.0;	// X1 RIGHT
		defCalib->Points[i].val[5] = 0.0;	// Y1 RIGHT
		defCalib->Points[i].val[6] = 10.0;	// X2 RIGHT
		defCalib->Points[i].val[7] = 10.0;	// Y2 RIGHT

		i=CALIB_TIG_AMPS_CMD;
		defCalib->Points[i].num = 4;

		defCalib->Points[i].val[0] = 0.0; 	// X1
		defCalib->Points[i].val[1] = 0.0; 	// Y1
		defCalib->Points[i].val[2] = 500.0; // X2
		defCalib->Points[i].val[3] = 500.0; // Y2

		i=CALIB_HW_AMPS_CMD;
		defCalib->Points[i].num = 4;

		defCalib->Points[i].val[0] = 0.0;	// X1
		defCalib->Points[i].val[1] = 0.0;	// Y1
		defCalib->Points[i].val[2] = 80.0; // X2  - 160 amp max
		defCalib->Points[i].val[3] = 80.0; // Y2

		i=CALIB_INDX_CMD;
		defCalib->Points[i].num = 4;

		defCalib->Points[i].val[0] = 0.0; 	// X1
		defCalib->Points[i].val[1] = 0.0; 	// Y1
		defCalib->Points[i].val[2] = 500.0; // X2
		defCalib->Points[i].val[3] = 500.0; // Y2

		//// How many calibrations we have
		defCalib->num = 8;
		//////////////////////////////////////////////////////////////////////////////////

		return 1;

}

///////////////////////////////////////////////////////////////
DINT  DefaultCalibr_SUPER_MINI(CurCalib_typ* defCalib){
UINT i;

		if(!defCalib)
			return 0;

		////////////////////////////////////////////////////////
		////   Default CALIBRATION

		i = CALIB_OSC_SFT_LIMIT;
		defCalib->Points[i].num = 4;

		defCalib->Points[i].val[0] = -1.0e+23;
		defCalib->Points[i].val[1] = 1.0e+23;
		defCalib->Points[i].val[2] = -1.0e+23;
		defCalib->Points[i].val[3] = 1.0e+23;

		i = CALIB_TIG_VOLT_FBK;
		defCalib->Points[i].num = 4;

		defCalib->Points[i].val[0] = 0.0; 	// 0 V
		defCalib->Points[i].val[1] = 1.44775391; 		// 6 V
		defCalib->Points[i].val[2] = 2.96142578; 		// 12 V
		defCalib->Points[i].val[3] = 4.45922852; 		// 18 V

		i = CALIB_TVL_SPEED_CMD;
		defCalib->Points[i].num = 8;

		// OMEGA 16 INCH  // 1"/min = 0.423 mm/s

		/*
		// Going Up
		defCalib->Points[i].val[0] = 0.846663; 	// X1 pos	 at 2"/min
		defCalib->Points[i].val[1] = 1.212983; 	// Y1 pos
		defCalib->Points[i].val[2] = 2.1166663; 	// X2 pos	at 5"/min
		defCalib->Points[i].val[3] = 2.621189; 	// Y2 pos

		// Going Down
		defCalib->Points[i].val[4] = 0.846663;		// X1 neg
		defCalib->Points[i].val[5] = 1.212983;		// Y1 neg
		defCalib->Points[i].val[6] = 2.1166663;	// X2 neg
		defCalib->Points[i].val[7] = 2.621189;	// Y2 neg
		*/

		defCalib->Points[i].val[0] = 0.0; 	// X1 pos	 at 2"/min
		defCalib->Points[i].val[1] = 0.0; 	// Y1 pos
		defCalib->Points[i].val[2] = 10.0; 	// X2 pos	at 5"/min
		defCalib->Points[i].val[3] = 10.0; 	// Y2 pos

		defCalib->Points[i].val[4] = 0.0;		// X1 neg
		defCalib->Points[i].val[5] = 0.0;		// Y1 neg
		defCalib->Points[i].val[6] = 10.0;	// X2 neg
		defCalib->Points[i].val[7] = 10.0;	// Y2 neg

		i = CALIB_WF_SPEED_CMD;
		defCalib->Points[i].num = 8;

		/*
		defCalib->Points[i].val[0] = 34.7; 	// X1 LEFT
		defCalib->Points[i].val[1] = 42.3; 	// Y1 LEFT
		defCalib->Points[i].val[2] = 70.6; 	// X2 LEFT
		defCalib->Points[i].val[3] = 84.7; 	// Y2 LEFT

		defCalib->Points[i].val[4] = 34.7;	// X1 RIGHT
		defCalib->Points[i].val[5] = 42.3;	// Y1 RIGHT
		defCalib->Points[i].val[6] = 70.6;	// X2 RIGHT
		defCalib->Points[i].val[7] = 84.7;	// Y2 RIGHT

		*/

		defCalib->Points[i].val[0] = 0.0; 	// X1 LEFT
		defCalib->Points[i].val[1] = 0.0; 	// Y1 LEFT
		defCalib->Points[i].val[2] = 10.0; 	// X2 LEFT
		defCalib->Points[i].val[3] = 10.0; 	// Y2 LEFT

		defCalib->Points[i].val[4] = 0.0;	// X1 RIGHT
		defCalib->Points[i].val[5] = 0.0;	// Y1 RIGHT
		defCalib->Points[i].val[6] = 10.0;	// X2 RIGHT
		defCalib->Points[i].val[7] = 10.0;	// Y2 RIGHT

		i = CALIB_WP_SPEED_CMD;
		defCalib->Points[i].num = 8;

		defCalib->Points[i].val[0] = 0.0;	// X1 LEFT
		defCalib->Points[i].val[1] = 0.0;	// Y1 LEFT
		defCalib->Points[i].val[2] = 10.0;	// X2 LEFT
		defCalib->Points[i].val[3] = 10.0;	// Y2 LEFT

		defCalib->Points[i].val[4] = 0.0;	// X1 RIGHT
		defCalib->Points[i].val[5] = 0.0;	// Y1 RIGHT
		defCalib->Points[i].val[6] = 10.0;	// X2 RIGHT
		defCalib->Points[i].val[7] = 10.0;	// Y2 RIGHT

		i=CALIB_TIG_AMPS_CMD;
		defCalib->Points[i].num = 4;
		/*
		defCalib->Points[i].val[0] = 92.0;	// X1
		defCalib->Points[i].val[1] = 80.0;	// Y1
		defCalib->Points[i].val[2] = 171.0; // X2
		defCalib->Points[i].val[3] = 150.0; // Y2
		defCalib->Points[i].num = 4;
		*/

		defCalib->Points[i].val[0] = 0.0; 	// X1
		defCalib->Points[i].val[1] = 0.0; 	// Y1
		defCalib->Points[i].val[2] = 500.0; // X2
		defCalib->Points[i].val[3] = 500.0; // Y2

		i=CALIB_HW_AMPS_CMD;
		defCalib->Points[i].num = 4;

		/*
		defCalib->Points[i].val[0] = 36.0;	// X1
		defCalib->Points[i].val[1] = 36.0;	// Y1
		defCalib->Points[i].val[2] = 83.0; // X2  - 160 amp max
		defCalib->Points[i].val[3] = 80.0; // Y2
		*/

		defCalib->Points[i].val[0] = 0.0;	// X1
		defCalib->Points[i].val[1] = 0.0;	// Y1
		defCalib->Points[i].val[2] = 80.0; // X2  - 160 amp max
		defCalib->Points[i].val[3] = 80.0; // Y2

		//// How many calibrations we have
		defCalib->num = 7;
		//////////////////////////////////////////////////////////////////////////////////

		return 1;

}

DINT DefaultCalibr_CLAMSHELL_HEAD(CurCalib_typ* defCalib){
UINT i;

		if(!defCalib)
			return 0;

		////////////////////////////////////////////////////////
		////   Default CALIBRATION

		i = CALIB_OSC_SFT_LIMIT;
		defCalib->Points[i].num = 4;

		defCalib->Points[i].val[0] = -1.0e+23;
		defCalib->Points[i].val[1] = 1.0e+23;
		defCalib->Points[i].val[2] = -1.0e+23;
		defCalib->Points[i].val[3] = 1.0e+23;

		i = CALIB_TIG_VOLT_FBK;
		defCalib->Points[i].num = 4;

		defCalib->Points[i].val[0] = 0.0; 	// 0 V
		defCalib->Points[i].val[1] = 1.44775391; 		// 6 V
		defCalib->Points[i].val[2] = 2.96142578; 		// 12 V
		defCalib->Points[i].val[3] = 4.45922852; 		// 18 V

		i = CALIB_TVL_SPEED_CMD;
		defCalib->Points[i].num = 8;

		// OMEGA 16 INCH  // 1"/min = 0.423 mm/s

		/*
		// Going Up
		defCalib->Points[i].val[0] = 0.846663; 	// X1 pos	 at 2"/min
		defCalib->Points[i].val[1] = 1.212983; 	// Y1 pos
		defCalib->Points[i].val[2] = 2.1166663; 	// X2 pos	at 5"/min
		defCalib->Points[i].val[3] = 2.621189; 	// Y2 pos

		// Going Down
		defCalib->Points[i].val[4] = 0.846663;		// X1 neg
		defCalib->Points[i].val[5] = 1.212983;		// Y1 neg
		defCalib->Points[i].val[6] = 2.1166663;	// X2 neg
		defCalib->Points[i].val[7] = 2.621189;	// Y2 neg
		*/

		defCalib->Points[i].val[0] = 0.0; 	// X1 pos	 at 2"/min
		defCalib->Points[i].val[1] = 0.0; 	// Y1 pos
		defCalib->Points[i].val[2] = 10.0; 	// X2 pos	at 5"/min
		defCalib->Points[i].val[3] = 10.0; 	// Y2 pos

		defCalib->Points[i].val[4] = 0.0;		// X1 neg
		defCalib->Points[i].val[5] = 0.0;		// Y1 neg
		defCalib->Points[i].val[6] = 10.0;	// X2 neg
		defCalib->Points[i].val[7] = 10.0;	// Y2 neg

		i = CALIB_WF_SPEED_CMD;
		defCalib->Points[i].num = 8;

		/*
		defCalib->Points[i].val[0] = 34.7; 	// X1 LEFT
		defCalib->Points[i].val[1] = 42.3; 	// Y1 LEFT
		defCalib->Points[i].val[2] = 70.6; 	// X2 LEFT
		defCalib->Points[i].val[3] = 84.7; 	// Y2 LEFT

		defCalib->Points[i].val[4] = 34.7;	// X1 RIGHT
		defCalib->Points[i].val[5] = 42.3;	// Y1 RIGHT
		defCalib->Points[i].val[6] = 70.6;	// X2 RIGHT
		defCalib->Points[i].val[7] = 84.7;	// Y2 RIGHT

		*/

		defCalib->Points[i].val[0] = 0.0; 	// X1 LEFT
		defCalib->Points[i].val[1] = 0.0; 	// Y1 LEFT
		defCalib->Points[i].val[2] = 10.0; 	// X2 LEFT
		defCalib->Points[i].val[3] = 10.0; 	// Y2 LEFT

		defCalib->Points[i].val[4] = 0.0;	// X1 RIGHT
		defCalib->Points[i].val[5] = 0.0;	// Y1 RIGHT
		defCalib->Points[i].val[6] = 10.0;	// X2 RIGHT
		defCalib->Points[i].val[7] = 10.0;	// Y2 RIGHT

		i = CALIB_WP_SPEED_CMD;
		defCalib->Points[i].num = 8;

		defCalib->Points[i].val[0] = 0.0;	// X1 LEFT
		defCalib->Points[i].val[1] = 0.0;	// Y1 LEFT
		defCalib->Points[i].val[2] = 10.0;	// X2 LEFT
		defCalib->Points[i].val[3] = 10.0;	// Y2 LEFT

		defCalib->Points[i].val[4] = 0.0;	// X1 RIGHT
		defCalib->Points[i].val[5] = 0.0;	// Y1 RIGHT
		defCalib->Points[i].val[6] = 10.0;	// X2 RIGHT
		defCalib->Points[i].val[7] = 10.0;	// Y2 RIGHT

		i=CALIB_TIG_AMPS_CMD;
		defCalib->Points[i].num = 4;
		/*
		defCalib->Points[i].val[0] = 92.0;	// X1
		defCalib->Points[i].val[1] = 80.0;	// Y1
		defCalib->Points[i].val[2] = 171.0; // X2
		defCalib->Points[i].val[3] = 150.0; // Y2
		defCalib->Points[i].num = 4;
		*/

		defCalib->Points[i].val[0] = 0.0; 	// X1
		defCalib->Points[i].val[1] = 0.0; 	// Y1
		defCalib->Points[i].val[2] = 500.0; // X2
		defCalib->Points[i].val[3] = 500.0; // Y2

		i=CALIB_HW_AMPS_CMD;
		defCalib->Points[i].num = 4;

		/*
		defCalib->Points[i].val[0] = 36.0;	// X1
		defCalib->Points[i].val[1] = 36.0;	// Y1
		defCalib->Points[i].val[2] = 83.0; // X2  - 160 amp max
		defCalib->Points[i].val[3] = 80.0; // Y2
		*/

		defCalib->Points[i].val[0] = 0.0;	// X1
		defCalib->Points[i].val[1] = 0.0;	// Y1
		defCalib->Points[i].val[2] = 80.0; // X2  - 160 amp max
		defCalib->Points[i].val[3] = 80.0; // Y2

		//// How many calibrations we have
		defCalib->num = 7;
		//////////////////////////////////////////////////////////////////////////////////

		return 1;

}
DINT DefaultCalibr_CHERRYPOINT_BPV2_HEAD(CurCalib_typ* defCalib){
UINT i;

		if(!defCalib)
			return 0;

		////////////////////////////////////////////////////////
		////   Default CALIBRATION

		i = CALIB_OSC_SFT_LIMIT;
		defCalib->Points[i].num = 4;

		defCalib->Points[i].val[0] = -1.0e+23;
		defCalib->Points[i].val[1] = 1.0e+23;
		defCalib->Points[i].val[2] = -1.0e+23;
		defCalib->Points[i].val[3] = 1.0e+23;

		i = CALIB_TIG_VOLT_FBK;
		defCalib->Points[i].num = 4;

		defCalib->Points[i].val[0] = 0.0; 	// 0 V
		defCalib->Points[i].val[1] = 1.44775391; 		// 6 V
		defCalib->Points[i].val[2] = 2.96142578; 		// 12 V
		defCalib->Points[i].val[3] = 4.45922852; 		// 18 V

		i = CALIB_TVL_SPEED_CMD;
		defCalib->Points[i].num = 8;

		// OMEGA 16 INCH  // 1"/min = 0.423 mm/s

		/*
		// Going Up
		defCalib->Points[i].val[0] = 0.846663; 	// X1 pos	 at 2"/min
		defCalib->Points[i].val[1] = 1.212983; 	// Y1 pos
		defCalib->Points[i].val[2] = 2.1166663; 	// X2 pos	at 5"/min
		defCalib->Points[i].val[3] = 2.621189; 	// Y2 pos

		// Going Down
		defCalib->Points[i].val[4] = 0.846663;		// X1 neg
		defCalib->Points[i].val[5] = 1.212983;		// Y1 neg
		defCalib->Points[i].val[6] = 2.1166663;	// X2 neg
		defCalib->Points[i].val[7] = 2.621189;	// Y2 neg
		*/

		defCalib->Points[i].val[0] = 0.0; 	// X1 pos	 at 2"/min
		defCalib->Points[i].val[1] = 0.0; 	// Y1 pos
		defCalib->Points[i].val[2] = 10.0; 	// X2 pos	at 5"/min
		defCalib->Points[i].val[3] = 10.0; 	// Y2 pos

		defCalib->Points[i].val[4] = 0.0;		// X1 neg
		defCalib->Points[i].val[5] = 0.0;		// Y1 neg
		defCalib->Points[i].val[6] = 10.0;	// X2 neg
		defCalib->Points[i].val[7] = 10.0;	// Y2 neg

		i = CALIB_WF_SPEED_CMD;
		defCalib->Points[i].num = 8;

		/*
		defCalib->Points[i].val[0] = 34.7; 	// X1 LEFT
		defCalib->Points[i].val[1] = 42.3; 	// Y1 LEFT
		defCalib->Points[i].val[2] = 70.6; 	// X2 LEFT
		defCalib->Points[i].val[3] = 84.7; 	// Y2 LEFT

		defCalib->Points[i].val[4] = 34.7;	// X1 RIGHT
		defCalib->Points[i].val[5] = 42.3;	// Y1 RIGHT
		defCalib->Points[i].val[6] = 70.6;	// X2 RIGHT
		defCalib->Points[i].val[7] = 84.7;	// Y2 RIGHT

		*/

		defCalib->Points[i].val[0] = 0.0; 	// X1 LEFT
		defCalib->Points[i].val[1] = 0.0; 	// Y1 LEFT
		defCalib->Points[i].val[2] = 10.0; 	// X2 LEFT
		defCalib->Points[i].val[3] = 10.0; 	// Y2 LEFT

		defCalib->Points[i].val[4] = 0.0;	// X1 RIGHT
		defCalib->Points[i].val[5] = 0.0;	// Y1 RIGHT
		defCalib->Points[i].val[6] = 10.0;	// X2 RIGHT
		defCalib->Points[i].val[7] = 10.0;	// Y2 RIGHT

		i = CALIB_WP_SPEED_CMD;
		defCalib->Points[i].num = 8;

		defCalib->Points[i].val[0] = 0.0;	// X1 LEFT
		defCalib->Points[i].val[1] = 0.0;	// Y1 LEFT
		defCalib->Points[i].val[2] = 10.0;	// X2 LEFT
		defCalib->Points[i].val[3] = 10.0;	// Y2 LEFT

		defCalib->Points[i].val[4] = 0.0;	// X1 RIGHT
		defCalib->Points[i].val[5] = 0.0;	// Y1 RIGHT
		defCalib->Points[i].val[6] = 10.0;	// X2 RIGHT
		defCalib->Points[i].val[7] = 10.0;	// Y2 RIGHT

		i=CALIB_TIG_AMPS_CMD;
		defCalib->Points[i].num = 4;
		/*
		defCalib->Points[i].val[0] = 92.0;	// X1
		defCalib->Points[i].val[1] = 80.0;	// Y1
		defCalib->Points[i].val[2] = 171.0; // X2
		defCalib->Points[i].val[3] = 150.0; // Y2
		defCalib->Points[i].num = 4;
		*/

		defCalib->Points[i].val[0] = 0.0; 	// X1
		defCalib->Points[i].val[1] = 0.0; 	// Y1
		defCalib->Points[i].val[2] = 500.0; // X2
		defCalib->Points[i].val[3] = 500.0; // Y2

		i=CALIB_HW_AMPS_CMD;
		defCalib->Points[i].num = 4;

		/*
		defCalib->Points[i].val[0] = 36.0;	// X1
		defCalib->Points[i].val[1] = 36.0;	// Y1
		defCalib->Points[i].val[2] = 83.0; // X2  - 160 amp max
		defCalib->Points[i].val[3] = 80.0; // Y2
		*/

		defCalib->Points[i].val[0] = 0.0;	// X1
		defCalib->Points[i].val[1] = 0.0;	// Y1
		defCalib->Points[i].val[2] = 80.0; // X2  - 160 amp max
		defCalib->Points[i].val[3] = 80.0; // Y2

		//// How many calibrations we have
		defCalib->num = 7;
		//////////////////////////////////////////////////////////////////////////////////

		return 1;

}

DINT DefaultCalibr_CHERRYPOINT_BPV1_HEAD(CurCalib_typ* defCalib){
UINT i;

		if(!defCalib)
			return 0;

		////////////////////////////////////////////////////////
		////   Default CALIBRATION

		i = CALIB_OSC_SFT_LIMIT;
		defCalib->Points[i].num = 4;

		defCalib->Points[i].val[0] = -1.0e+23;
		defCalib->Points[i].val[1] = 1.0e+23;
		defCalib->Points[i].val[2] = -1.0e+23;
		defCalib->Points[i].val[3] = 1.0e+23;

		i = CALIB_TIG_VOLT_FBK;
		defCalib->Points[i].num = 4;

		defCalib->Points[i].val[0] = 0.0; 	// 0 V
		defCalib->Points[i].val[1] = 1.44775391; 		// 6 V
		defCalib->Points[i].val[2] = 2.96142578; 		// 12 V
		defCalib->Points[i].val[3] = 4.45922852; 		// 18 V

		i = CALIB_TVL_SPEED_CMD;
		defCalib->Points[i].num = 8;

		// OMEGA 16 INCH  // 1"/min = 0.423 mm/s

		/*
		// Going Up
		defCalib->Points[i].val[0] = 0.846663; 	// X1 pos	 at 2"/min
		defCalib->Points[i].val[1] = 1.212983; 	// Y1 pos
		defCalib->Points[i].val[2] = 2.1166663; 	// X2 pos	at 5"/min
		defCalib->Points[i].val[3] = 2.621189; 	// Y2 pos

		// Going Down
		defCalib->Points[i].val[4] = 0.846663;		// X1 neg
		defCalib->Points[i].val[5] = 1.212983;		// Y1 neg
		defCalib->Points[i].val[6] = 2.1166663;	// X2 neg
		defCalib->Points[i].val[7] = 2.621189;	// Y2 neg
		*/

		defCalib->Points[i].val[0] = 0.0; 	// X1 pos	 at 2"/min
		defCalib->Points[i].val[1] = 0.0; 	// Y1 pos
		defCalib->Points[i].val[2] = 10.0; 	// X2 pos	at 5"/min
		defCalib->Points[i].val[3] = 10.0; 	// Y2 pos

		defCalib->Points[i].val[4] = 0.0;		// X1 neg
		defCalib->Points[i].val[5] = 0.0;		// Y1 neg
		defCalib->Points[i].val[6] = 10.0;	// X2 neg
		defCalib->Points[i].val[7] = 10.0;	// Y2 neg

		i = CALIB_WF_SPEED_CMD;
		defCalib->Points[i].num = 8;

		/*
		defCalib->Points[i].val[0] = 34.7; 	// X1 LEFT
		defCalib->Points[i].val[1] = 42.3; 	// Y1 LEFT
		defCalib->Points[i].val[2] = 70.6; 	// X2 LEFT
		defCalib->Points[i].val[3] = 84.7; 	// Y2 LEFT

		defCalib->Points[i].val[4] = 34.7;	// X1 RIGHT
		defCalib->Points[i].val[5] = 42.3;	// Y1 RIGHT
		defCalib->Points[i].val[6] = 70.6;	// X2 RIGHT
		defCalib->Points[i].val[7] = 84.7;	// Y2 RIGHT

		*/

		defCalib->Points[i].val[0] = 0.0; 	// X1 LEFT
		defCalib->Points[i].val[1] = 0.0; 	// Y1 LEFT
		defCalib->Points[i].val[2] = 10.0; 	// X2 LEFT
		defCalib->Points[i].val[3] = 10.0; 	// Y2 LEFT

		defCalib->Points[i].val[4] = 0.0;	// X1 RIGHT
		defCalib->Points[i].val[5] = 0.0;	// Y1 RIGHT
		defCalib->Points[i].val[6] = 10.0;	// X2 RIGHT
		defCalib->Points[i].val[7] = 10.0;	// Y2 RIGHT

		i = CALIB_WP_SPEED_CMD;
		defCalib->Points[i].num = 8;

		defCalib->Points[i].val[0] = 0.0;	// X1 LEFT
		defCalib->Points[i].val[1] = 0.0;	// Y1 LEFT
		defCalib->Points[i].val[2] = 10.0;	// X2 LEFT
		defCalib->Points[i].val[3] = 10.0;	// Y2 LEFT

		defCalib->Points[i].val[4] = 0.0;	// X1 RIGHT
		defCalib->Points[i].val[5] = 0.0;	// Y1 RIGHT
		defCalib->Points[i].val[6] = 10.0;	// X2 RIGHT
		defCalib->Points[i].val[7] = 10.0;	// Y2 RIGHT

		i=CALIB_TIG_AMPS_CMD;
		defCalib->Points[i].num = 4;
		/*
		defCalib->Points[i].val[0] = 92.0;	// X1
		defCalib->Points[i].val[1] = 80.0;	// Y1
		defCalib->Points[i].val[2] = 171.0; // X2
		defCalib->Points[i].val[3] = 150.0; // Y2
		defCalib->Points[i].num = 4;
		*/

		defCalib->Points[i].val[0] = 0.0; 	// X1
		defCalib->Points[i].val[1] = 0.0; 	// Y1
		defCalib->Points[i].val[2] = 500.0; // X2
		defCalib->Points[i].val[3] = 500.0; // Y2

		i=CALIB_HW_AMPS_CMD;
		defCalib->Points[i].num = 4;

		/*
		defCalib->Points[i].val[0] = 36.0;	// X1
		defCalib->Points[i].val[1] = 36.0;	// Y1
		defCalib->Points[i].val[2] = 83.0; // X2  - 160 amp max
		defCalib->Points[i].val[3] = 80.0; // Y2
		*/

		defCalib->Points[i].val[0] = 0.0;	// X1
		defCalib->Points[i].val[1] = 0.0;	// Y1
		defCalib->Points[i].val[2] = 80.0; // X2  - 160 amp max
		defCalib->Points[i].val[3] = 80.0; // Y2

		//// How many calibrations we have
		defCalib->num = 7;
		//////////////////////////////////////////////////////////////////////////////////

		return 1;

}

DINT  DefaultCalibr_BPV_F_HEAD(CurCalib_typ* defCalib){
UINT i;

		if(!defCalib)
			return 0;

		////////////////////////////////////////////////////////
		////   Default CALIBRATION

		i = CALIB_OSC_SFT_LIMIT;
		defCalib->Points[i].num = 4;

		defCalib->Points[i].val[0] = -1.0e+23;
		defCalib->Points[i].val[1] = 1.0e+23;
		defCalib->Points[i].val[2] = -1.0e+23;
		defCalib->Points[i].val[3] = 1.0e+23;

		i = CALIB_TIG_VOLT_FBK;
		defCalib->Points[i].num = 4;

		defCalib->Points[i].val[0] = 0.0; 	// 0 V
		defCalib->Points[i].val[1] = 1.44775391; 		// 6 V
		defCalib->Points[i].val[2] = 2.96142578; 		// 12 V
		defCalib->Points[i].val[3] = 4.45922852; 		// 18 V

		i = CALIB_TVL_SPEED_CMD;
		defCalib->Points[i].num = 8;

		// OMEGA 16 INCH  // 1"/min = 0.423 mm/s

		/*
		// Going Up
		defCalib->Points[i].val[0] = 0.846663; 	// X1 pos	 at 2"/min
		defCalib->Points[i].val[1] = 1.212983; 	// Y1 pos
		defCalib->Points[i].val[2] = 2.1166663; 	// X2 pos	at 5"/min
		defCalib->Points[i].val[3] = 2.621189; 	// Y2 pos

		// Going Down
		defCalib->Points[i].val[4] = 0.846663;		// X1 neg
		defCalib->Points[i].val[5] = 1.212983;		// Y1 neg
		defCalib->Points[i].val[6] = 2.1166663;	// X2 neg
		defCalib->Points[i].val[7] = 2.621189;	// Y2 neg
		*/

		defCalib->Points[i].val[0] = 0.0; 	// X1 pos	 at 2"/min
		defCalib->Points[i].val[1] = 0.0; 	// Y1 pos
		defCalib->Points[i].val[2] = 10.0; 	// X2 pos	at 5"/min
		defCalib->Points[i].val[3] = 10.0; 	// Y2 pos

		defCalib->Points[i].val[4] = 0.0;		// X1 neg
		defCalib->Points[i].val[5] = 0.0;		// Y1 neg
		defCalib->Points[i].val[6] = 10.0;	// X2 neg
		defCalib->Points[i].val[7] = 10.0;	// Y2 neg

		i = CALIB_WF_SPEED_CMD;
		defCalib->Points[i].num = 8;

		/*
		defCalib->Points[i].val[0] = 34.7; 	// X1 LEFT
		defCalib->Points[i].val[1] = 42.3; 	// Y1 LEFT
		defCalib->Points[i].val[2] = 70.6; 	// X2 LEFT
		defCalib->Points[i].val[3] = 84.7; 	// Y2 LEFT

		defCalib->Points[i].val[4] = 34.7;	// X1 RIGHT
		defCalib->Points[i].val[5] = 42.3;	// Y1 RIGHT
		defCalib->Points[i].val[6] = 70.6;	// X2 RIGHT
		defCalib->Points[i].val[7] = 84.7;	// Y2 RIGHT

		*/

		defCalib->Points[i].val[0] = 0.0; 	// X1 LEFT
		defCalib->Points[i].val[1] = 0.0; 	// Y1 LEFT
		defCalib->Points[i].val[2] = 10.0; 	// X2 LEFT
		defCalib->Points[i].val[3] = 10.0; 	// Y2 LEFT

		defCalib->Points[i].val[4] = 0.0;	// X1 RIGHT
		defCalib->Points[i].val[5] = 0.0;	// Y1 RIGHT
		defCalib->Points[i].val[6] = 10.0;	// X2 RIGHT
		defCalib->Points[i].val[7] = 10.0;	// Y2 RIGHT

		i = CALIB_WP_SPEED_CMD;
		defCalib->Points[i].num = 8;

		defCalib->Points[i].val[0] = 0.0;	// X1 LEFT
		defCalib->Points[i].val[1] = 0.0;	// Y1 LEFT
		defCalib->Points[i].val[2] = 10.0;	// X2 LEFT
		defCalib->Points[i].val[3] = 10.0;	// Y2 LEFT

		defCalib->Points[i].val[4] = 0.0;	// X1 RIGHT
		defCalib->Points[i].val[5] = 0.0;	// Y1 RIGHT
		defCalib->Points[i].val[6] = 10.0;	// X2 RIGHT
		defCalib->Points[i].val[7] = 10.0;	// Y2 RIGHT

		i=CALIB_TIG_AMPS_CMD;
		defCalib->Points[i].num = 4;
		/*
		defCalib->Points[i].val[0] = 92.0;	// X1
		defCalib->Points[i].val[1] = 80.0;	// Y1
		defCalib->Points[i].val[2] = 171.0; // X2
		defCalib->Points[i].val[3] = 150.0; // Y2
		defCalib->Points[i].num = 4;
		*/

		defCalib->Points[i].val[0] = 0.0; 	// X1
		defCalib->Points[i].val[1] = 0.0; 	// Y1
		defCalib->Points[i].val[2] = 500.0; // X2
		defCalib->Points[i].val[3] = 500.0; // Y2

		i=CALIB_HW_AMPS_CMD;
		defCalib->Points[i].num = 4;

		/*
		defCalib->Points[i].val[0] = 36.0;	// X1
		defCalib->Points[i].val[1] = 36.0;	// Y1
		defCalib->Points[i].val[2] = 83.0; // X2  - 160 amp max
		defCalib->Points[i].val[3] = 80.0; // Y2
		*/

		defCalib->Points[i].val[0] = 0.0;	// X1
		defCalib->Points[i].val[1] = 0.0;	// Y1
		defCalib->Points[i].val[2] = 80.0; // X2  - 160 amp max
		defCalib->Points[i].val[3] = 80.0; // Y2

		//// How many calibrations we have
		defCalib->num = 7;
		//////////////////////////////////////////////////////////////////////////////////

		return 1;

}

DINT  DefaultCalibr_BPV_V1_MT(CurCalib_typ* defCalib){
UINT i;

		if(!defCalib)
			return 0;

		////////////////////////////////////////////////////////
		////   Default CALIBRATION

		i = CALIB_OSC_SFT_LIMIT;
		defCalib->Points[i].num = 4;

		defCalib->Points[i].val[0] = -1.0e+23;
		defCalib->Points[i].val[1] = 1.0e+23;
		defCalib->Points[i].val[2] = -1.0e+23;
		defCalib->Points[i].val[3] = 1.0e+23;

		i = CALIB_TIG_VOLT_FBK;
		defCalib->Points[i].num = 4;

		defCalib->Points[i].val[0] = 0.0; 	// 0 V
		defCalib->Points[i].val[1] = 1.44775391; 		// 6 V
		defCalib->Points[i].val[2] = 2.96142578; 		// 12 V
		defCalib->Points[i].val[3] = 4.45922852; 		// 18 V

		i = CALIB_TVL_SPEED_CMD;
		defCalib->Points[i].num = 8;

		// OMEGA 16 INCH  // 1"/min = 0.423 mm/s

		/*
		// Going Up
		defCalib->Points[i].val[0] = 0.846663; 	// X1 pos	 at 2"/min
		defCalib->Points[i].val[1] = 1.212983; 	// Y1 pos
		defCalib->Points[i].val[2] = 2.1166663; 	// X2 pos	at 5"/min
		defCalib->Points[i].val[3] = 2.621189; 	// Y2 pos

		// Going Down
		defCalib->Points[i].val[4] = 0.846663;		// X1 neg
		defCalib->Points[i].val[5] = 1.212983;		// Y1 neg
		defCalib->Points[i].val[6] = 2.1166663;	// X2 neg
		defCalib->Points[i].val[7] = 2.621189;	// Y2 neg
		*/

		defCalib->Points[i].val[0] = 0.0; 	// X1 pos	 at 2"/min
		defCalib->Points[i].val[1] = 0.0; 	// Y1 pos
		defCalib->Points[i].val[2] = 10.0; 	// X2 pos	at 5"/min
		defCalib->Points[i].val[3] = 10.0; 	// Y2 pos

		defCalib->Points[i].val[4] = 0.0;		// X1 neg
		defCalib->Points[i].val[5] = 0.0;		// Y1 neg
		defCalib->Points[i].val[6] = 10.0;	// X2 neg
		defCalib->Points[i].val[7] = 10.0;	// Y2 neg

		i = CALIB_WF_SPEED_CMD;
		defCalib->Points[i].num = 8;

		/*
		defCalib->Points[i].val[0] = 34.7; 	// X1 LEFT
		defCalib->Points[i].val[1] = 42.3; 	// Y1 LEFT
		defCalib->Points[i].val[2] = 70.6; 	// X2 LEFT
		defCalib->Points[i].val[3] = 84.7; 	// Y2 LEFT

		defCalib->Points[i].val[4] = 34.7;	// X1 RIGHT
		defCalib->Points[i].val[5] = 42.3;	// Y1 RIGHT
		defCalib->Points[i].val[6] = 70.6;	// X2 RIGHT
		defCalib->Points[i].val[7] = 84.7;	// Y2 RIGHT

		*/

		defCalib->Points[i].val[0] = 0.0; 	// X1 LEFT
		defCalib->Points[i].val[1] = 0.0; 	// Y1 LEFT
		defCalib->Points[i].val[2] = 10.0; 	// X2 LEFT
		defCalib->Points[i].val[3] = 10.0; 	// Y2 LEFT

		defCalib->Points[i].val[4] = 0.0;	// X1 RIGHT
		defCalib->Points[i].val[5] = 0.0;	// Y1 RIGHT
		defCalib->Points[i].val[6] = 10.0;	// X2 RIGHT
		defCalib->Points[i].val[7] = 10.0;	// Y2 RIGHT

		i = CALIB_WP_SPEED_CMD;
		defCalib->Points[i].num = 8;

		defCalib->Points[i].val[0] = 0.0;	// X1 LEFT
		defCalib->Points[i].val[1] = 0.0;	// Y1 LEFT
		defCalib->Points[i].val[2] = 10.0;	// X2 LEFT
		defCalib->Points[i].val[3] = 10.0;	// Y2 LEFT

		defCalib->Points[i].val[4] = 0.0;	// X1 RIGHT
		defCalib->Points[i].val[5] = 0.0;	// Y1 RIGHT
		defCalib->Points[i].val[6] = 10.0;	// X2 RIGHT
		defCalib->Points[i].val[7] = 10.0;	// Y2 RIGHT

		i=CALIB_TIG_AMPS_CMD;
		defCalib->Points[i].num = 4;
		/*
		defCalib->Points[i].val[0] = 92.0;	// X1
		defCalib->Points[i].val[1] = 80.0;	// Y1
		defCalib->Points[i].val[2] = 171.0; // X2
		defCalib->Points[i].val[3] = 150.0; // Y2
		defCalib->Points[i].num = 4;
		*/

		defCalib->Points[i].val[0] = 0.0; 	// X1
		defCalib->Points[i].val[1] = 0.0; 	// Y1
		defCalib->Points[i].val[2] = 500.0; // X2
		defCalib->Points[i].val[3] = 500.0; // Y2

		i=CALIB_HW_AMPS_CMD;
		defCalib->Points[i].num = 4;

		/*
		defCalib->Points[i].val[0] = 36.0;	// X1
		defCalib->Points[i].val[1] = 36.0;	// Y1
		defCalib->Points[i].val[2] = 83.0; // X2  - 160 amp max
		defCalib->Points[i].val[3] = 80.0; // Y2
		*/

		defCalib->Points[i].val[0] = 0.0;	// X1
		defCalib->Points[i].val[1] = 0.0;	// Y1
		defCalib->Points[i].val[2] = 80.0; // X2  - 160 amp max
		defCalib->Points[i].val[3] = 80.0; // Y2

		//// How many calibrations we have
		defCalib->num = 7;
		//////////////////////////////////////////////////////////////////////////////////

		return 1;

}

DINT  DefaultCalibr_M_94(CurCalib_typ* defCalib){
UINT i;

		if(!defCalib)
			return 0;

		////////////////////////////////////////////////////////
		////   Default CALIBRATION

		i = CALIB_OSC_SFT_LIMIT;
		defCalib->Points[i].num = 4;

		defCalib->Points[i].val[0] = -1.0e+23;
		defCalib->Points[i].val[1] = 1.0e+23;
		defCalib->Points[i].val[2] = -1.0e+23;
		defCalib->Points[i].val[3] = 1.0e+23;

		i = CALIB_TIG_VOLT_FBK;
		defCalib->Points[i].num = 4;

		defCalib->Points[i].val[0] = 0.0; 	// 0 V
		defCalib->Points[i].val[1] = 1.44775391; 		// 6 V
		defCalib->Points[i].val[2] = 2.96142578; 		// 12 V
		defCalib->Points[i].val[3] = 4.45922852; 		// 18 V

		i = CALIB_TVL_SPEED_CMD;
		defCalib->Points[i].num = 8;

		// OMEGA 16 INCH  // 1"/min = 0.423 mm/s

		/*
		// Going Up
		defCalib->Points[i].val[0] = 0.846663; 	// X1 pos	 at 2"/min
		defCalib->Points[i].val[1] = 1.212983; 	// Y1 pos
		defCalib->Points[i].val[2] = 2.1166663; 	// X2 pos	at 5"/min
		defCalib->Points[i].val[3] = 2.621189; 	// Y2 pos

		// Going Down
		defCalib->Points[i].val[4] = 0.846663;		// X1 neg
		defCalib->Points[i].val[5] = 1.212983;		// Y1 neg
		defCalib->Points[i].val[6] = 2.1166663;	// X2 neg
		defCalib->Points[i].val[7] = 2.621189;	// Y2 neg
		*/

		defCalib->Points[i].val[0] = 0.0; 	// X1 pos	 at 2"/min
		defCalib->Points[i].val[1] = 0.0; 	// Y1 pos
		defCalib->Points[i].val[2] = 10.0; 	// X2 pos	at 5"/min
		defCalib->Points[i].val[3] = 10.0; 	// Y2 pos

		defCalib->Points[i].val[4] = 0.0;		// X1 neg
		defCalib->Points[i].val[5] = 0.0;		// Y1 neg
		defCalib->Points[i].val[6] = 10.0;	// X2 neg
		defCalib->Points[i].val[7] = 10.0;	// Y2 neg

		i = CALIB_WF_SPEED_CMD;
		defCalib->Points[i].num = 8;

		/*
		defCalib->Points[i].val[0] = 34.7; 	// X1 LEFT
		defCalib->Points[i].val[1] = 42.3; 	// Y1 LEFT
		defCalib->Points[i].val[2] = 70.6; 	// X2 LEFT
		defCalib->Points[i].val[3] = 84.7; 	// Y2 LEFT

		defCalib->Points[i].val[4] = 34.7;	// X1 RIGHT
		defCalib->Points[i].val[5] = 42.3;	// Y1 RIGHT
		defCalib->Points[i].val[6] = 70.6;	// X2 RIGHT
		defCalib->Points[i].val[7] = 84.7;	// Y2 RIGHT

		*/

		defCalib->Points[i].val[0] = 0.0; 	// X1 LEFT
		defCalib->Points[i].val[1] = 0.0; 	// Y1 LEFT
		defCalib->Points[i].val[2] = 10.0; 	// X2 LEFT
		defCalib->Points[i].val[3] = 10.0; 	// Y2 LEFT

		defCalib->Points[i].val[4] = 0.0;	// X1 RIGHT
		defCalib->Points[i].val[5] = 0.0;	// Y1 RIGHT
		defCalib->Points[i].val[6] = 10.0;	// X2 RIGHT
		defCalib->Points[i].val[7] = 10.0;	// Y2 RIGHT

		i = CALIB_WP_SPEED_CMD;
		defCalib->Points[i].num = 8;

		defCalib->Points[i].val[0] = 0.0;	// X1 LEFT
		defCalib->Points[i].val[1] = 0.0;	// Y1 LEFT
		defCalib->Points[i].val[2] = 10.0;	// X2 LEFT
		defCalib->Points[i].val[3] = 10.0;	// Y2 LEFT
```
